KUKA KRL program: MyProgram_122().src

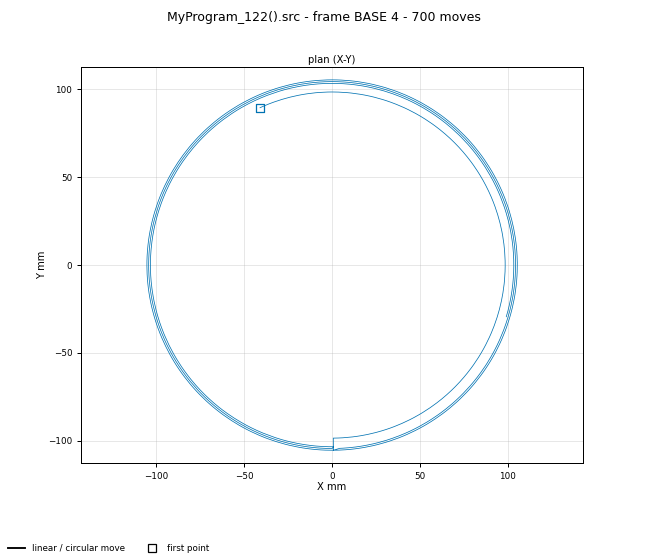
[picture p0: tool path of MyProgram_122().src in frame BASE 4, 700 of 700 moves have a stored position in this frame; points joined in program order, loops and branches not executed]
&ACCESS RVP
&REL 1
&PARAM TEMPLATE = C:\KRC\Roboter\Template\vorgabe
&PARAM EDITMASK = *
DEF MyProgram_122()
; ---- Setting reference (Base) ----
$BASE = BASE_DATA[4]

; --------------------------
; ---- Setting tool (TCP) ----
$TOOL = TOOL_DATA[3]
; --------------------------

$VEL.CP = VEL_APROX_PRINT
Startdeposition()
$VEL.CP = VEL_PRINT
LIN {X -40.9948,Y 89.481,Z 102,A 109.215,B 24.9184,C -2.0865,E1 24.9347,E2 -23.8628} C_DIS
LIN {X -38.5849,Y 90.5452,Z 102,A 107.7654,B 24.918,C -2.0917,E1 24.9383,E2 -22.4221} C_DIS
LIN {X -36.007,Y 91.6,Z 102,A 106.0596,B 24.918,C -2.091,E1 24.9428,E2 -20.711} C_DIS
LIN {X -33.1406,Y 92.6775,Z 102,A 104.2606,B 24.9179,C -2.0927,E1 24.9475,E2 -18.9123} C_DIS
LIN {X -30.6483,Y 93.5301,Z 102,A 102.9444,B 24.9171,C -2.1021,E1 24.9509,E2 -17.616} C_DIS
LIN {X -28.5659,Y 94.1882,Z 102,A 101.5499,B 24.9174,C -2.0993,E1 24.9547,E2 -16.2123} C_DIS
LIN {X -26.2518,Y 94.8593,Z 102,A 100.0341,B 24.9175,C -2.0968,E1 24.9588,E2 -14.6883} C_DIS
LIN {X -23.9044,Y 95.4778,Z 102,A 98.6262,B 24.9175,C -2.0984,E1 24.9626,E2 -13.2821} C_DIS
LIN {X -21.3156,Y 96.0877,Z 102,A 97.2954,B 24.9167,C -2.1074,E1 24.9661,E2 -11.9709} C_DIS
LIN {X -19.1831,Y 96.5372,Z 102,A 95.8048,B 24.9172,C -2.1007,E1 24.9703,E2 -10.4627} C_DIS
LIN {X -16.8179,Y 96.9772,Z 102,A 94.4012,B 24.9172,C -2.1016,E1 24.9741,E2 -9.06} C_DIS
LIN {X -14.1942,Y 97.3947,Z 102,A 92.9697,B 24.9168,C -2.1067,E1 24.978,E2 -7.6393} C_DIS
LIN {X -11.6809,Y 97.7276,Z 102,A 91.4888,B 24.9168,C -2.1075,E1 24.9821,E2 -6.159} C_DIS
LIN {X -9.5679,Y 97.9582,Z 102,A 90.1489,B 24.9169,C -2.1045,E1 24.9859,E2 -4.8112} C_DIS
LIN {X -7.202,Y 98.1607,Z 102,A 88.8601,B 24.9166,C -2.1084,E1 24.9895,E2 -3.5312} C_DIS
LIN {X -4.6001,Y 98.3161,Z 102,A 87.3398,B 24.9166,C -2.1088,E1 24.9937,E2 -2.0116} C_DIS
LIN {X -2.4401,Y 98.3944,Z 102,A 85.9895,B 24.9168,C -2.1059,E1 24.9975,E2 -0.6542} C_DIS
LIN {X -0.0607,Y 98.4244,Z 102,A 84.6864,B 24.9166,C -2.1091,E1 25.0011,E2 0.6413} C_DIS
LIN {X 3.6137,Y 98.3584,Z 102,A 82.4028,B 24.917,C -2.1042,E1 25.0075,E2 2.9361} C_DIS
LIN {X 6.3319,Y 98.2195,Z 102,A 81.0916,B 24.9162,C -2.1141,E1 25.0111,E2 4.2236} C_DIS
LIN {X 8.7012,Y 98.0382,Z 102,A 79.7032,B 24.9162,C -2.1138,E1 25.015,E2 5.6119} C_DIS
LIN {X 10.8611,Y 97.8236,Z 102,A 78.2118,B 24.9169,C -2.1054,E1 25.0191,E2 7.1222} C_DIS
LIN {X 13.4885,Y 97.4949,Z 102,A 76.8979,B 24.9162,C -2.1133,E1 25.0227,E2 8.4164} C_DIS
LIN {X 15.8676,Y 97.1361,Z 102,A 75.4989,B 24.9162,C -2.1129,E1 25.0266,E2 9.8148} C_DIS
LIN {X 18.2378,Y 96.7192,Z 102,A 73.8857,B 24.9169,C -2.1047,E1 25.0311,E2 11.4458} C_DIS
LIN {X 21.5808,Y 96.0296,Z 102,A 71.8924,B 24.917,C -2.1035,E1 25.0365,E2 13.4393} C_DIS
LIN {X 23.9252,Y 95.4726,Z 102,A 70.491,B 24.917,C -2.1027,E1 25.0403,E2 14.8406} C_DIS
LIN {X 26.4725,Y 94.7967,Z 102,A 69.0598,B 24.9169,C -2.1055,E1 25.0441,E2 16.2629} C_DIS
LIN {X 28.7857,Y 94.1201,Z 102,A 67.7784,B 24.9166,C -2.1089,E1 25.0476,E2 17.5339} C_DIS
LIN {X 30.9879,Y 93.4187,Z 102,A 66.2645,B 24.9172,C -2.1016,E1 25.0516,E2 19.0622} C_DIS
LIN {X 33.3777,Y 92.5912,Z 102,A 64.7955,B 24.9172,C -2.1004,E1 25.0555,E2 20.531} C_DIS
LIN {X 36.5486,Y 91.3873,Z 102,A 62.8757,B 24.9172,C -2.1004,E1 25.0605,E2 22.4465} C_DIS
LIN {X 38.7951,Y 90.4564,Z 102,A 61.3644,B 24.9177,C -2.0954,E1 25.0644,E2 23.9662} C_DIS
LIN {X 40.9951,Y 89.4809,Z 102,A 59.9392,B 24.9179,C -2.0929,E1 25.068,E2 25.3938} C_DIS
LIN {X 43.3728,Y 88.3516,Z 102,A 58.5388,B 24.9176,C -2.096,E1 25.0715,E2 26.7832} C_DIS
LIN {X 45.637,Y 87.2032,Z 102,A 57.1115,B 24.9176,C -2.096,E1 25.075,E2 28.2067} C_DIS
LIN {X 47.4644,Y 86.2239,Z 102,A 55.7597,B 24.9182,C -2.0889,E1 25.0784,E2 29.5713} C_DIS
LIN {X 50.0077,Y 84.7721,Z 102,A 54.0718,B 24.9183,C -2.0871,E1 25.0825,E2 31.2584} C_DIS
LIN {X 52.7518,Y 83.0937,Z 102,A 52.3478,B 24.9181,C -2.0898,E1 25.0865,E2 32.9706} C_DIS
LIN {X 54.8752,Y 81.7063,Z 102,A 50.9442,B 24.9181,C -2.0901,E1 25.0898,E2 34.3687} C_DIS
LIN {X 56.6984,Y 80.453,Z 102,A 49.5558,B 24.9185,C -2.0842,E1 25.093,E2 35.7664} C_DIS
LIN {X 58.6281,Y 79.058,Z 102,A 47.9451,B 24.9194,C -2.0733,E1 25.0967,E2 37.3971} C_DIS
LIN {X 61.4921,Y 76.8514,Z 102,A 45.8467,B 24.9197,C -2.0697,E1 25.1013,E2 39.4962} C_DIS
LIN {X 64.2951,Y 74.5223,Z 102,A 43.7362,B 24.92,C -2.066,E1 25.1058,E2 41.6072} C_DIS
LIN {X 66.9924,Y 72.1072,Z 102,A 41.6381,B 24.9203,C -2.0621,E1 25.1101,E2 43.7061} C_DIS
LIN {X 69.5959,Y 69.5978,Z 102,A 39.5415,B 24.9206,C -2.058,E1 25.1143,E2 45.8037} C_DIS
LIN {X 72.1053,Y 66.9944,Z 102,A 37.4476,B 24.9209,C -2.0537,E1 25.1183,E2 47.8985} C_DIS
LIN {X 74.5277,Y 64.2888,Z 102,A 35.3391,B 24.9213,C -2.0491,E1 25.1222,E2 50.0084} C_DIS
LIN {X 76.8501,Y 61.4937,Z 102,A 33.2405,B 24.9216,C -2.0448,E1 25.1259,E2 52.1075} C_DIS
LIN {X 79.0559,Y 58.631,Z 102,A 31.2593,B 24.9216,C -2.0443,E1 25.1292,E2 54.0804} C_DIS
LIN {X 80.4674,Y 56.6783,Z 102,A 29.6553,B 24.9225,C -2.033,E1 25.1318,E2 55.7032} C_DIS
LIN {X 82.6251,Y 53.4819,Z 102,A 27.8533,B 24.9216,C -2.0444,E1 25.1345,E2 57.4694} C_DIS
LIN {X 84.0971,Y 51.1345,Z 102,A 26.0418,B 24.9225,C -2.0325,E1 25.1372,E2 59.2998} C_DIS
LIN {X 85.7558,Y 48.3027,Z 102,A 24.1231,B 24.923,C -2.027,E1 25.1399,E2 61.2215} C_DIS
LIN {X 87.367,Y 45.326,Z 102,A 22.0924,B 24.9235,C -2.0192,E1 25.1426,E2 63.26} C_DIS
LIN {X 89.0655,Y 41.8874,Z 102,A 19.9181,B 24.9239,C -2.0152,E1 25.1452,E2 65.432} C_DIS
LIN {X 90.4636,Y 38.7786,Z 102,A 17.9782,B 24.9242,C -2.0112,E1 25.1474,E2 67.3707} C_DIS
LIN {X 91.6025,Y 36.0009,Z 102,A 16.2585,B 24.9245,C -2.0073,E1 25.1492,E2 69.0903} C_DIS
LIN {X 92.6741,Y 33.1502,Z 102,A 14.4811,B 24.9249,C -2.0018,E1 25.1509,E2 70.8706} C_DIS
LIN {X 93.5274,Y 30.6569,Z 102,A 13.1779,B 24.9245,C -2.0063,E1 25.152,E2 72.1558} C_DIS
LIN {X 94.1858,Y 28.574,Z 102,A 11.7748,B 24.9252,C -1.9973,E1 25.1532,E2 73.5722} C_DIS
LIN {X 94.8669,Y 26.2236,Z 102,A 10.2814,B 24.9257,C -1.9902,E1 25.1544,E2 75.0737} C_DIS
LIN {X 95.4791,Y 23.8988,Z 102,A 8.8903,B 24.926,C -1.9863,E1 25.1553,E2 76.4662} C_DIS
LIN {X 96.0936,Y 21.2884,Z 102,A 7.5866,B 24.9256,C -1.9916,E1 25.1561,E2 77.7497} C_DIS
LIN {X 96.5329,Y 19.2052,Z 102,A 6.0876,B 24.9267,C -1.9775,E1 25.157,E2 79.2733} C_DIS
LIN {X 96.9811,Y 16.795,Z 102,A 4.6967,B 24.9269,C -1.9744,E1 25.1577,E2 80.6632} C_DIS
LIN {X 97.3996,Y 14.1594,Z 102,A 3.3975,B 24.9265,C -1.9796,E1 25.1582,E2 81.9427} C_DIS
LIN {X 97.7073,Y 11.8542,Z 102,A 1.8366,B 24.9275,C -1.9671,E1 25.1588,E2 83.5237} C_DIS
LIN {X 98.1077,Y 7.8712,Z 102,A -0.4988,B 24.928,C -1.9595,E1 25.1594,E2 85.8633} C_DIS
LIN {X 98.316,Y 4.602,Z 102,A -2.3059,B 24.9282,C -1.9573,E1 25.1596,E2 87.6648} C_DIS
LIN {X 98.3951,Y 2.4176,Z 102,A -3.5706,B 24.9285,C -1.9535,E1 25.1598,E2 88.931} C_DIS
LIN {X 98.4213,Y -0.5653,Z 102,A -5.399,B 24.9291,C -1.9443,E1 25.1598,E2 90.7702} C_DIS
LIN {X 98.3552,Y -3.6891,Z 102,A -7.192,B 24.9295,C -1.9394,E1 25.1596,E2 92.564} C_DIS
LIN {X 98.2215,Y -6.3023,Z 102,A -8.4936,B 24.9292,C -1.9433,E1 25.1594,E2 93.8488} C_DIS
LIN {X 98.0389,Y -8.6932,Z 102,A -9.8785,B 24.9295,C -1.9392,E1 25.1591,E2 95.2351} C_DIS
LIN {X 97.8239,Y -10.8585,Z 102,A -11.3563,B 24.9304,C -1.9267,E1 25.1587,E2 96.7336} C_DIS
LIN {X 97.4984,Y -13.4641,Z 102,A -12.7946,B 24.9305,C -1.9254,E1 25.1582,E2 98.1666} C_DIS
LIN {X 97.1354,Y -15.8721,Z 102,A -14.0618,B 24.9305,C -1.9268,E1 25.1576,E2 99.423} C_DIS
LIN {X 96.7189,Y -18.2393,Z 102,A -15.5914,B 24.9311,C -1.9171,E1 25.1568,E2 100.9665} C_DIS
LIN {X 96.2873,Y -20.4005,Z 102,A -16.8444,B 24.9313,C -1.9142,E1 25.1561,E2 102.2191} C_DIS
LIN {X 95.7064,Y -22.9672,Z 102,A -18.2464,B 24.9313,C -1.9144,E1 25.1553,E2 103.6124} C_DIS
LIN {X 95.1162,Y -25.3005,Z 102,A -19.7578,B 24.9319,C -1.9056,E1 25.1542,E2 105.1358} C_DIS
LIN {X 94.4693,Y -27.6185,Z 102,A -21.1492,B 24.9322,C -1.9016,E1 25.1531,E2 106.5289} C_DIS
LIN {X 93.827,Y -29.731,Z 102,A -22.4266,B 24.9325,C -1.8978,E1 25.1521,E2 107.8078} C_DIS
LIN {X 92.9958,Y -32.2334,Z 102,A -23.9518,B 24.9328,C -1.8934,E1 25.1507,E2 109.3347} C_DIS
LIN {X 92.1626,Y -34.5434,Z 102,A -25.3693,B 24.9331,C -1.8895,E1 25.1493,E2 110.7536} C_DIS
LIN {X 91.3772,Y -36.5734,Z 102,A -26.6278,B 24.9333,C -1.8859,E1 25.1481,E2 112.0136} C_DIS
LIN {X 90.4568,Y -38.7942,Z 102,A -28.1186,B 24.9339,C -1.878,E1 25.1464,E2 113.5149} C_DIS
LIN {X 89.4819,Y -40.9929,Z 102,A -29.5106,B 24.9342,C -1.8741,E1 25.1448,E2 114.9085} C_DIS
LIN {X 88.3535,Y -43.3691,Z 102,A -30.9312,B 24.9342,C -1.8738,E1 25.1431,E2 116.3221} C_DIS
LIN {X 87.372,Y -45.3161,Z 102,A -32.2879,B 24.9347,C -1.8666,E1 25.1414,E2 117.6886} C_DIS
LIN {X 86.239,Y -47.4367,Z 102,A -33.6741,B 24.9349,C -1.863,E1 25.1395,E2 119.0761} C_DIS
LIN {X 84.9241,Y -49.7506,Z 102,A -35.2558,B 24.9353,C -1.8573,E1 25.1373,E2 120.6632} C_DIS
LIN {X 83.1402,Y -52.6793,Z 102,A -37.1049,B 24.9353,C -1.8573,E1 25.1346,E2 122.5028} C_DIS
LIN {X 81.7038,Y -54.8789,Z 102,A -38.5066,B 24.9353,C -1.858,E1 25.1324,E2 123.8958} C_DIS
LIN {X 80.4701,Y -56.6745,Z 102,A -39.8888,B 24.9358,C -1.85,E1 25.1302,E2 125.2902} C_DIS
LIN {X 79.0513,Y -58.6372,Z 102,A -41.503,B 24.9367,C -1.8382,E1 25.1275,E2 126.9245} C_DIS
LIN {X 76.8441,Y -61.5014,Z 102,A -43.4664,B 24.9367,C -1.8381,E1 25.1242,E2 128.8789} C_DIS
LIN {X 74.8272,Y -63.9373,Z 102,A -45.3366,B 24.9371,C -1.8321,E1 25.1208,E2 130.7546} C_DIS
LIN {X 72.5141,Y -66.5491,Z 102,A -47.3417,B 24.9374,C -1.828,E1 25.117,E2 132.7606} C_DIS
LIN {X 70.0204,Y -69.168,Z 102,A -49.3744,B 24.9375,C -1.8256,E1 25.1131,E2 134.7902} C_DIS
LIN {X 67.8252,Y -71.324,Z 102,A -51.305,B 24.9382,C -1.8158,E1 25.1092,E2 136.7358} C_DIS
LIN {X 65.2036,Y -73.7287,Z 102,A -53.3867,B 24.9386,C -1.8106,E1 25.1049,E2 138.8215} C_DIS
LIN {X 62.4378,Y -76.0852,Z 102,A -55.4885,B 24.9388,C -1.8063,E1 25.1003,E2 140.9253} C_DIS
LIN {X 59.5809,Y -78.3424,Z 102,A -57.5598,B 24.939,C -1.8036,E1 25.0958,E2 142.9953} C_DIS
LIN {X 57.4689,Y -79.9033,Z 102,A -58.9038,B 24.9388,C -1.8076,E1 25.0928,E2 144.3253} C_DIS
LIN {X 55.688,Y -81.1559,Z 102,A -60.2643,B 24.9392,C -1.8014,E1 25.0896,E2 145.6957} C_DIS
LIN {X 53.4819,Y -82.6251,Z 102,A -61.5838,B 24.9388,C -1.807,E1 25.0866,E2 146.9977} C_DIS
LIN {X 51.4301,Y -83.9176,Z 102,A -63.0217,B 24.939,C -1.8033,E1 25.0832,E2 148.4397} C_DIS
LIN {X 49.5184,Y -85.0606,Z 102,A -64.6107,B 24.94,C -1.7897,E1 25.0793,E2 150.0559} C_DIS
LIN {X 46.3754,Y -86.8143,Z 102,A -66.4863,B 24.9396,C -1.7944,E1 25.0747,E2 151.915} C_DIS
LIN {X 44.2425,Y -87.9205,Z 102,A -67.88,B 24.9398,C -1.7923,E1 25.0713,E2 153.3099} C_DIS
LIN {X 41.8786,Y -89.0696,Z 102,A -69.2882,B 24.9396,C -1.7945,E1 25.0677,E2 154.7093} C_DIS
LIN {X 39.6914,Y -90.0656,Z 102,A -70.8131,B 24.9401,C -1.7875,E1 25.0638,E2 156.2468} C_DIS
LIN {X 37.4486,Y -91.0209,Z 102,A -72.0962,B 24.9399,C -1.7906,E1 25.0606,E2 157.5196} C_DIS
LIN {X 35.4186,Y -91.8311,Z 102,A -73.4851,B 24.9403,C -1.7844,E1 25.0569,E2 158.9201} C_DIS
LIN {X 33.1106,Y -92.688,Z 102,A -75.0087,B 24.9407,C -1.7791,E1 25.0529,E2 160.453} C_DIS
LIN {X 30.6275,Y -93.5369,Z 102,A -76.318,B 24.9403,C -1.7854,E1 25.0495,E2 161.7448} C_DIS
LIN {X 28.004,Y -94.3549,Z 102,A -78.1162,B 24.9409,C -1.7761,E1 25.0446,E2 163.5618} C_DIS
LIN {X 24.8626,Y -95.2316,Z 102,A -79.8055,B 24.9405,C -1.7819,E1 25.0401,E2 165.2347} C_DIS
LIN {X 22.4912,Y -95.8193,Z 102,A -81.3437,B 24.9409,C -1.7762,E1 25.0359,E2 166.7843} C_DIS
LIN {X 20.3694,Y -96.2938,Z 102,A -82.8131,B 24.9415,C -1.7674,E1 25.0318,E2 168.2725} C_DIS
LIN {X 16.7828,Y -96.9831,Z 102,A -84.826,B 24.9413,C -1.7699,E1 25.0263,E2 170.2772} C_DIS
LIN {X 14.4201,Y -97.3626,Z 102,A -86.1187,B 24.9411,C -1.7726,E1 25.0228,E2 171.5623} C_DIS
LIN {X 11.5691,Y -97.7407,Z 102,A -87.6865,B 24.9409,C -1.7755,E1 25.0185,E2 173.122} C_DIS
LIN {X 8.2496,Y -98.0774,Z 102,A -89.6312,B 24.9409,C -1.7744,E1 25.0131,E2 175.0683} C_DIS
LIN {X 6.0869,Y -98.2361,Z 102,A -91.0704,B 24.9415,C -1.7673,E1 25.009,E2 176.5236} C_DIS
LIN {X 3.3973,Y -98.365,Z 102,A -92.4427,B 24.941,C -1.7739,E1 25.0052,E2 177.8798} C_DIS
LIN {X 0.6801,Y -98.4206,Z 102,A -93.8704,B 24.9407,C -1.7791,E1 25.0013,E2 179.295} C_DIS
Enddeposition()
LIN {X 0.7313,Y -105.3176,Z 103,A -93.556,B 24.9473,C -1.6774,E1 25.0015,E2 179.2217} C_DIS
Startdeposition()
$VEL.CP = VEL_PRINT
LIN {X -1.2925,Y -105.3149,Z 103,A -94.9939,B 24.9481,C -1.6637,E1 24.9974,E2 180.692} C_DIS
LIN {X -3.7589,Y -105.2551,Z 103,A -96.3407,B 24.9481,C -1.6634,E1 24.9936,E2 182.0398} C_DIS
LIN {X -6.3408,Y -105.1311,Z 103,A -97.7467,B 24.9481,C -1.6634,E1 24.9897,E2 183.4464} C_DIS
LIN {X -8.919,Y -104.9438,Z 103,A -99.1478,B 24.9481,C -1.6636,E1 24.9858,E2 184.8475} C_DIS
LIN {X -11.6089,Y -104.6811,Z 103,A -100.6185,B 24.9481,C -1.6636,E1 24.9817,E2 186.3187} C_DIS
LIN {X -14.1744,Y -104.3647,Z 103,A -102.0255,B 24.9481,C -1.6639,E1 24.9778,E2 187.7262} C_DIS
LIN {X -16.7314,Y -103.9854,Z 103,A -103.4327,B 24.9481,C -1.6642,E1 24.9739,E2 189.1339} C_DIS
LIN {X -19.2783,Y -103.5434,Z 103,A -104.8397,B 24.9481,C -1.6647,E1 24.9701,E2 190.5412} C_DIS
LIN {X -21.8136,Y -103.0391,Z 103,A -106.2476,B 24.9481,C -1.6652,E1 24.9662,E2 191.9495} C_DIS
LIN {X -24.2209,Y -102.4993,Z 103,A -107.5961,B 24.9481,C -1.6656,E1 24.9625,E2 193.2988} C_DIS
LIN {X -26.729,Y -101.874,Z 103,A -108.9991,B 24.948,C -1.6666,E1 24.9587,E2 194.7015} C_DIS
LIN {X -29.2211,Y -101.1874,Z 103,A -110.4124,B 24.948,C -1.6672,E1 24.9549,E2 196.1156} C_DIS
LIN {X -31.6604,Y -100.4507,Z 103,A -111.804,B 24.9479,C -1.668,E1 24.9512,E2 197.5077} C_DIS
LIN {X -34.2626,Y -99.594,Z 103,A -113.2888,B 24.9478,C -1.6694,E1 24.9473,E2 198.9919} C_DIS
LIN {X -36.5857,Y -98.7636,Z 103,A -114.6335,B 24.9478,C -1.6705,E1 24.9438,E2 200.3367} C_DIS
LIN {X -38.9985,Y -97.836,Z 103,A -116.0427,B 24.9476,C -1.6718,E1 24.9401,E2 201.746} C_DIS
LIN {X -41.3878,Y -96.8494,Z 103,A -117.4487,B 24.9476,C -1.6733,E1 24.9365,E2 203.1518} C_DIS
LIN {X -43.8595,Y -95.7561,Z 103,A -118.926,B 24.9474,C -1.6746,E1 24.9327,E2 204.6294} C_DIS
LIN {X -46.0901,Y -94.702,Z 103,A -120.2766,B 24.9474,C -1.6759,E1 24.9293,E2 205.9804} C_DIS
LIN {X -48.4003,Y -93.5423,Z 103,A -121.6818,B 24.9473,C -1.6777,E1 24.9258,E2 207.385} C_DIS
LIN {X -50.6814,Y -92.3263,Z 103,A -123.0919,B 24.9471,C -1.6794,E1 24.9223,E2 208.7951} C_DIS
LIN {X -52.9319,Y -91.0548,Z 103,A -124.5028,B 24.9471,C -1.6812,E1 24.9189,E2 210.2059} C_DIS
LIN {X -55.1506,Y -89.7283,Z 103,A -125.9134,B 24.9469,C -1.6832,E1 24.9156,E2 211.6163} C_DIS
LIN {X -57.3091,Y -88.3651,Z 103,A -127.3087,B 24.9468,C -1.6851,E1 24.9123,E2 213.0115} C_DIS
LIN {X -59.5845,Y -86.8481,Z 103,A -128.8,B 24.9466,C -1.6873,E1 24.9088,E2 214.5024} C_DIS
LIN {X -61.602,Y -85.4281,Z 103,A -130.1469,B 24.9466,C -1.6894,E1 24.9058,E2 215.849} C_DIS
LIN {X -63.6799,Y -83.8906,Z 103,A -131.5635,B 24.9464,C -1.6915,E1 24.9026,E2 217.2657} C_DIS
LIN {X -65.7195,Y -82.3025,Z 103,A -132.9703,B 24.9462,C -1.694,E1 24.8995,E2 218.6716} C_DIS
LIN {X -67.7195,Y -80.6649,Z 103,A -134.3826,B 24.9461,C -1.6965,E1 24.8965,E2 220.0835} C_DIS
LIN {X -69.6787,Y -78.9787,Z 103,A -135.7996,B 24.9459,C -1.6988,E1 24.8935,E2 221.5005} C_DIS
LIN {X -71.6828,Y -77.1652,Z 103,A -137.2715,B 24.9457,C -1.7017,E1 24.8905,E2 222.9715} C_DIS
LIN {X -73.555,Y -75.3828,Z 103,A -138.684,B 24.9456,C -1.7044,E1 24.8876,E2 224.3835} C_DIS
LIN {X -75.3,Y -73.6388,Z 103,A -140.0112,B 24.9453,C -1.7078,E1 24.885,E2 225.7082} C_DIS
LIN {X -77.0845,Y -71.7687,Z 103,A -141.4455,B 24.9453,C -1.7099,E1 24.8823,E2 227.1438} C_DIS
LIN {X -78.8226,Y -69.8553,Z 103,A -142.8635,B 24.945,C -1.7126,E1 24.8796,E2 228.5617} C_DIS
LIN {X -80.5896,Y -67.8102,Z 103,A -144.3363,B 24.9448,C -1.7159,E1 24.877,E2 230.0333} C_DIS
LIN {X -82.2294,Y -65.812,Z 103,A -145.7499,B 24.9446,C -1.7189,E1 24.8745,E2 231.4463} C_DIS
LIN {X -83.6473,Y -63.998,Z 103,A -147.0343,B 24.9446,C -1.7208,E1 24.8723,E2 232.7323} C_DIS
LIN {X -85.3596,Y -61.6979,Z 103,A -148.5772,B 24.9442,C -1.7253,E1 24.8697,E2 234.2721} C_DIS
LIN {X -86.8481,Y -59.5845,Z 103,A -149.9913,B 24.944,C -1.7285,E1 24.8675,E2 235.6853} C_DIS
LIN {X -88.2842,Y -57.4352,Z 103,A -151.4054,B 24.9438,C -1.7319,E1 24.8653,E2 237.0986} C_DIS
LIN {X -89.6671,Y -55.2513,Z 103,A -152.8199,B 24.9436,C -1.7352,E1 24.8632,E2 238.5122} C_DIS
LIN {X -90.9961,Y -53.0341,Z 103,A -154.2342,B 24.9433,C -1.7387,E1 24.8612,E2 239.9256} C_DIS
LIN {X -92.2702,Y -50.785,Z 103,A -155.6485,B 24.9431,C -1.7422,E1 24.8593,E2 241.3389} C_DIS
LIN {X -93.4887,Y -48.5052,Z 103,A -157.0636,B 24.9429,C -1.7458,E1 24.8574,E2 242.7532} C_DIS
LIN {X -94.5986,Y -46.3019,Z 103,A -158.3982,B 24.9426,C -1.7498,E1 24.8558,E2 244.0853} C_DIS
LIN {X -95.7561,Y -43.8595,Z 103,A -159.8931,B 24.9424,C -1.753,E1 24.854,E2 245.5806} C_DIS
LIN {X -96.7566,Y -41.6044,Z 103,A -161.2487,B 24.9422,C -1.7564,E1 24.8525,E2 246.9356} C_DIS
LIN {X -97.7929,Y -39.1082,Z 103,A -162.7234,B 24.9419,C -1.7605,E1 24.8509,E2 248.4088} C_DIS
LIN {X -99.1661,Y -35.4822,Z 103,A -164.8465,B 24.9415,C -1.7662,E1 24.8489,E2 250.5302} C_DIS
LIN {X -99.9693,Y -33.1495,Z 103,A -166.1975,B 24.9413,C -1.7699,E1 24.8477,E2 251.88} C_DIS
LIN {X -100.7876,Y -30.5736,Z 103,A -167.6771,B 24.941,C -1.774,E1 24.8464,E2 253.3585} C_DIS
LIN {X -101.5076,Y -28.0909,Z 103,A -169.0929,B 24.9408,C -1.778,E1 24.8454,E2 254.773} C_DIS
LIN {X -102.4448,Y -24.4502,Z 103,A -171.157,B 24.9404,C -1.7836,E1 24.844,E2 256.8358} C_DIS
LIN {X -103.014,Y -21.9287,Z 103,A -172.5495,B 24.94,C -1.7885,E1 24.8431,E2 258.2249} C_DIS
LIN {X -103.706,Y -18.3741,Z 103,A -174.5824,B 24.9398,C -1.7924,E1 24.8421,E2 260.2604} C_DIS
LIN {X -104.1649,Y -15.5705,Z 103,A -176.1126,B 24.9394,C -1.7978,E1 24.8414,E2 261.7869} C_DIS
LIN {X -104.5156,Y -13.0095,Z 103,A -177.5287,B 24.9391,C -1.8019,E1 24.8409,E2 263.2017} C_DIS
LIN {X -104.8034,Y -10.4406,Z 103,A -178.9447,B 24.9389,C -1.806,E1 24.8405,E2 264.6162} C_DIS
LIN {X -105.0374,Y -7.748,Z 103,A 179.5798,B 24.9386,C -1.8105,E1 24.8402,E2 266.0899} C_DIS
LIN {X -105.196,Y -5.1679,Z 103,A 178.1638,B 24.9383,C -1.8147,E1 24.8399,E2 267.5045} C_DIS
LIN {X -105.2911,Y -2.5848,Z 103,A 176.7475,B 24.938,C -1.8189,E1 24.8399,E2 268.9193} C_DIS
LIN {X -105.3199,Y -0.4985,Z 103,A 175.5316,B 24.938,C -1.8197,E1 24.8398,E2 270.1407} C_DIS
LIN {X -105.2946,Y 2.394,Z 103,A 174.0149,B 24.9374,C -1.8268,E1 24.8398,E2 271.6496} C_DIS
LIN {X -105.196,Y 5.1679,Z 103,A 172.4989,B 24.9371,C -1.8314,E1 24.84,E2 273.1637} C_DIS
LIN {X -105.0374,Y 7.748,Z 103,A 171.083,B 24.9368,C -1.8356,E1 24.8403,E2 274.5781} C_DIS
LIN {X -104.7054,Y 11.3769,Z 103,A 169.0769,B 24.9365,C -1.8412,E1 24.8408,E2 276.5829} C_DIS
LIN {X -104.3647,Y 14.1744,Z 103,A 167.5426,B 24.9361,C -1.8461,E1 24.8414,E2 278.1147} C_DIS
LIN {X -104.0034,Y 16.6149,Z 103,A 166.1908,B 24.9358,C -1.8501,E1 24.8419,E2 279.465} C_DIS
LIN {X -103.5434,Y 19.2783,Z 103,A 164.7104,B 24.9355,C -1.8544,E1 24.8427,E2 280.9438} C_DIS
LIN {X -103.0391,Y 21.8136,Z 103,A 163.294,B 24.9352,C -1.8585,E1 24.8435,E2 282.3587} C_DIS
LIN {X -102.4993,Y 24.2209,Z 103,A 161.9772,B 24.9349,C -1.8637,E1 24.8443,E2 283.6709} C_DIS
LIN {X -101.5383,Y 27.9772,Z 103,A 159.8433,B 24.9345,C -1.8696,E1 24.8458,E2 285.8034} C_DIS
LIN {X -100.8212,Y 30.4606,Z 103,A 158.3975,B 24.9343,C -1.8726,E1 24.8469,E2 287.2503} C_DIS
LIN {X -100.007,Y 33.0378,Z 103,A 156.9221,B 24.934,C -1.877,E1 24.8482,E2 288.7235} C_DIS
LIN {X -99.2051,Y 35.371,Z 103,A 155.5659,B 24.9337,C -1.8807,E1 24.8495,E2 290.0787} C_DIS
LIN {X -98.2654,Y 37.9052,Z 103,A 154.0907,B 24.9334,C -1.885,E1 24.8509,E2 291.5518} C_DIS
LIN {X -97.3056,Y 40.3053,Z 103,A 152.675,B 24.9331,C -1.889,E1 24.8524,E2 292.9659} C_DIS
LIN {X -96.2871,Y 42.6812,Z 103,A 151.2592,B 24.9328,C -1.8929,E1 24.854,E2 294.3802} C_DIS
LIN {X -95.2604,Y 44.9245,Z 103,A 149.9034,B 24.9326,C -1.8965,E1 24.8556,E2 295.7348} C_DIS
LIN {X -94.0769,Y 47.3543,Z 103,A 148.4286,B 24.9323,C -1.9007,E1 24.8574,E2 297.2076} C_DIS
LIN {X -92.9413,Y 49.5446,Z 103,A 147.0725,B 24.932,C -1.9042,E1 24.8591,E2 298.5626} C_DIS
LIN {X -91.6975,Y 51.8105,Z 103,A 145.6575,B 24.9318,C -1.908,E1 24.8611,E2 299.976} C_DIS
LIN {X -90.3384,Y 54.1467,Z 103,A 144.183,B 24.9315,C -1.912,E1 24.8632,E2 301.4485} C_DIS
LIN {X -88.9824,Y 56.3475,Z 103,A 142.7677,B 24.9312,C -1.9157,E1 24.8652,E2 302.8622} C_DIS
LIN {X -87.6376,Y 58.4158,Z 103,A 141.4175,B 24.9309,C -1.9192,E1 24.8673,E2 304.2109} C_DIS
LIN {X -86.1103,Y 60.6457,Z 103,A 139.9381,B 24.9307,C -1.9229,E1 24.8697,E2 305.6887} C_DIS
LIN {X -84.6657,Y 62.6457,Z 103,A 138.588,B 24.9304,C -1.9263,E1 24.8719,E2 307.0373} C_DIS
LIN {X -83.0588,Y 64.7616,Z 103,A 137.1355,B 24.9302,C -1.9299,E1 24.8744,E2 308.4882} C_DIS
LIN {X -81.4898,Y 66.7245,Z 103,A 135.7592,B 24.9299,C -1.9332,E1 24.8768,E2 309.8631} C_DIS
LIN {X -79.8278,Y 68.7043,Z 103,A 134.3402,B 24.9297,C -1.9363,E1 24.8793,E2 311.281} C_DIS
LIN {X -78.0391,Y 70.7305,Z 103,A 132.8663,B 24.9294,C -1.9399,E1 24.8821,E2 312.7528} C_DIS
LIN {X -76.2797,Y 72.6243,Z 103,A 131.4527,B 24.9292,C -1.9432,E1 24.8848,E2 314.165} C_DIS
LIN {X -74.4745,Y 74.4745,Z 103,A 130.039,B 24.929,C -1.9463,E1 24.8875,E2 315.5772} C_DIS
LIN {X -72.7092,Y 76.198,Z 103,A 128.6899,B 24.9288,C -1.9493,E1 24.8903,E2 316.9248} C_DIS
LIN {X -70.8173,Y 77.9594,Z 103,A 127.2766,B 24.9285,C -1.9523,E1 24.8932,E2 318.3367} C_DIS
LIN {X -68.8831,Y 79.6736,Z 103,A 125.8585,B 24.9283,C -1.955,E1 24.8961,E2 319.7538} C_DIS
LIN {X -66.9545,Y 81.3006,Z 103,A 124.4838,B 24.9281,C -1.958,E1 24.8991,E2 321.1267} C_DIS
LIN {X -64.7979,Y 83.0309,Z 103,A 122.9728,B 24.9279,C -1.961,E1 24.9024,E2 322.6362} C_DIS
LIN {X -62.7407,Y 84.5961,Z 103,A 121.5602,B 24.9277,C -1.9637,E1 24.9055,E2 324.0474} C_DIS
LIN {X -60.6457,Y 86.1103,Z 103,A 120.1477,B 24.9275,C -1.9663,E1 24.9087,E2 325.4585} C_DIS
LIN {X -57.6507,Y 88.1421,Z 103,A 118.1487,B 24.9273,C -1.9691,E1 24.9134,E2 327.4576} C_DIS
LIN {X -55.3512,Y 89.6047,Z 103,A 116.6768,B 24.9271,C -1.9723,E1 24.9169,E2 328.9266} C_DIS
LIN {X -53.3457,Y 90.8119,Z 103,A 115.3635,B 24.9271,C -1.9731,E1 24.92,E2 330.2418} C_DIS
LIN {X -50.785,Y 92.2702,Z 103,A 113.7942,B 24.9267,C -1.9772,E1 24.9238,E2 331.8062} C_DIS
LIN {X -48.5052,Y 93.4887,Z 103,A 112.3824,B 24.9265,C -1.9793,E1 24.9273,E2 333.2167} C_DIS
LIN {X -46.3019,Y 94.5986,Z 103,A 111.0489,B 24.9264,C -1.9818,E1 24.9306,E2 334.5479} C_DIS
LIN {X -43.8595,Y 95.7561,Z 103,A 109.5605,B 24.9262,C -1.9834,E1 24.9344,E2 336.0362} C_DIS
LIN {X -41.4963,Y 96.8037,Z 103,A 108.1497,B 24.9262,C -1.9853,E1 24.938,E2 337.4459} C_DIS
LIN {X -39.1082,Y 97.7929,Z 103,A 106.7391,B 24.926,C -1.9871,E1 24.9417,E2 338.8553} C_DIS
LIN {X -36.6964,Y 98.7232,Z 103,A 105.3289,B 24.9258,C -1.9888,E1 24.9453,E2 340.2643} C_DIS
LIN {X -34.2626,Y 99.594,Z 103,A 103.9188,B 24.9258,C -1.9904,E1 24.949,E2 341.6734} C_DIS
LIN {X -31.9202,Y 100.3686,Z 103,A 102.5682,B 24.9256,C -1.9917,E1 24.9526,E2 343.0234} C_DIS
LIN {X -29.4474,Y 101.1217,Z 103,A 101.172,B 24.9255,C -1.9936,E1 24.9564,E2 344.4173} C_DIS
LIN {X -26.8432,Y 101.8447,Z 103,A 99.6899,B 24.9254,C -1.9947,E1 24.9604,E2 345.8992} C_DIS
LIN {X -24.4502,Y 102.4448,Z 103,A 98.3754,B 24.9252,C -1.997,E1 24.9639,E2 347.21} C_DIS
LIN {X -21.9287,Y 103.014,Z 103,A 96.9361,B 24.9252,C -1.997,E1 24.9678,E2 348.6511} C_DIS
LIN {X -19.394,Y 103.5212,Z 103,A 95.5273,B 24.9252,C -1.9981,E1 24.9717,E2 350.059} C_DIS
LIN {X -16.7314,Y 103.9854,Z 103,A 94.0547,B 24.9251,C -1.999,E1 24.9757,E2 351.5307} C_DIS
LIN {X -14.1744,Y 104.3647,Z 103,A 92.6465,B 24.9251,C -1.9999,E1 24.9796,E2 352.938} C_DIS
LIN {X -11.6089,Y 104.6811,Z 103,A 91.2386,B 24.925,C -2.0006,E1 24.9835,E2 354.3451} C_DIS
LIN {X -8.1224,Y 105.0075,Z 103,A 89.3002,B 24.925,C -2.0003,E1 24.9889,E2 356.2852} C_DIS
LIN {X -5.1679,Y 105.196,Z 103,A 87.7195,B 24.9249,C -2.002,E1 24.9933,E2 357.8623} C_DIS
LIN {X -2.8306,Y 105.2835,Z 103,A 86.435,B 24.9249,C -2.002,E1 24.9969,E2 359.1471} C_DIS
LIN {X -0.1178,Y 105.3221,Z 103,A 84.9645,B 24.9249,C -2.0024,E1 25.001,E2 360.6165} C_DIS
LIN {X 2.5848,Y 105.2911,Z 103,A 83.4989,B 24.9248,C -2.0028,E1 25.0051,E2 362.0809} C_DIS
LIN {X 5.1679,Y 105.196,Z 103,A 82.0921,B 24.9248,C -2.0028,E1 25.009,E2 363.4872} C_DIS
LIN {X 7.748,Y 105.0374,Z 103,A 80.6859,B 24.9248,C -2.0028,E1 25.013,E2 364.8929} C_DIS
LIN {X 10.2061,Y 104.8265,Z 103,A 79.339,B 24.9248,C -2.0025,E1 25.0167,E2 366.2397} C_DIS
LIN {X 12.601,Y 104.5649,Z 103,A 78.0251,B 24.9248,C -2.0022,E1 25.0203,E2 367.5534} C_DIS
LIN {X 15.3374,Y 104.1994,Z 103,A 76.528,B 24.9248,C -2.002,E1 25.0245,E2 369.0497} C_DIS
LIN {X 18.0062,Y 103.7722,Z 103,A 75.0638,B 24.9248,C -2.0017,E1 25.0285,E2 370.5131} C_DIS
LIN {X 20.4318,Y 103.3213,Z 103,A 73.7178,B 24.9249,C -2.001,E1 25.0322,E2 371.8592} C_DIS
LIN {X 23.0764,Y 102.7637,Z 103,A 72.2541,B 24.9249,C -2.0005,E1 25.0362,E2 373.3221} C_DIS
LIN {X 25.5914,Y 102.1664,Z 103,A 70.8496,B 24.925,C -1.9998,E1 25.04,E2 374.7263} C_DIS
LIN {X 27.9772,Y 101.5383,Z 103,A 69.5043,B 24.925,C -1.9988,E1 25.0436,E2 376.0718} C_DIS
LIN {X 30.4606,Y 100.8212,Z 103,A 68.1265,B 24.925,C -1.9989,E1 25.0473,E2 377.447} C_DIS
LIN {X 33.0378,Y 100.007,Z 103,A 66.6375,B 24.9252,C -1.997,E1 25.0513,E2 378.9378} C_DIS
LIN {X 35.371,Y 99.2051,Z 103,A 65.2979,B 24.9253,C -1.9959,E1 25.0548,E2 380.2772} C_DIS
LIN {X 37.795,Y 98.3072,Z 103,A 63.8897,B 24.9254,C -1.9945,E1 25.0585,E2 381.6857} C_DIS
LIN {X 41.3878,Y 96.8494,Z 103,A 61.7851,B 24.9256,C -1.9925,E1 25.0639,E2 383.7903} C_DIS
LIN {X 43.7521,Y 95.8045,Z 103,A 60.3873,B 24.9256,C -1.9912,E1 25.0675,E2 385.1876} C_DIS
LIN {X 46.0901,Y 94.702,Z 103,A 58.9798,B 24.9258,C -1.9894,E1 25.071,E2 386.5956} C_DIS
LIN {X 48.5052,Y 93.4887,Z 103,A 57.5187,B 24.9259,C -1.9879,E1 25.0747,E2 388.0564} C_DIS
LIN {X 50.785,Y 92.2702,Z 103,A 56.1166,B 24.926,C -1.9861,E1 25.0781,E2 389.4586} C_DIS
LIN {X 53.0341,Y 90.9961,Z 103,A 54.7145,B 24.9262,C -1.9843,E1 25.0815,E2 390.8609} C_DIS
LIN {X 54.8577,Y 89.9063,Z 103,A 53.5023,B 24.9265,C -1.9803,E1 25.0844,E2 392.0787} C_DIS
LIN {X 57.336,Y 88.3478,Z 103,A 51.9752,B 24.9265,C -1.9804,E1 25.088,E2 393.6005} C_DIS
LIN {X 59.5845,Y 86.8481,Z 103,A 50.5101,B 24.9266,C -1.9782,E1 25.0914,E2 395.066} C_DIS
LIN {X 61.602,Y 85.4281,Z 103,A 49.1729,B 24.9268,C -1.9761,E1 25.0944,E2 396.4034} C_DIS
LIN {X 63.6799,Y 83.8906,Z 103,A 47.8027,B 24.9268,C -1.9751,E1 25.0975,E2 397.7711} C_DIS
LIN {X 65.812,Y 82.2294,Z 103,A 46.3078,B 24.9271,C -1.9714,E1 25.1008,E2 399.2693} C_DIS
LIN {X 67.7195,Y 80.6649,Z 103,A 44.9711,B 24.9273,C -1.9691,E1 25.1036,E2 400.6063} C_DIS
LIN {X 69.6788,Y 78.9787,Z 103,A 43.5657,B 24.9275,C -1.9663,E1 25.1066,E2 402.0127} C_DIS
LIN {X 71.6828,Y 77.1652,Z 103,A 42.107,B 24.9277,C -1.9638,E1 25.1096,E2 403.4714} C_DIS
LIN {X 73.555,Y 75.3828,Z 103,A 40.707,B 24.9279,C -1.9611,E1 25.1124,E2 404.872} C_DIS
LIN {X 75.3,Y 73.6388,Z 103,A 39.3824,B 24.9281,C -1.959,E1 25.115,E2 406.196} C_DIS
LIN {X 77.0845,Y 71.7686,Z 103,A 37.9666,B 24.9283,C -1.9555,E1 25.1177,E2 407.6139} C_DIS
LIN {X 78.8226,Y 69.8553,Z 103,A 36.5957,B 24.9284,C -1.9537,E1 25.1203,E2 408.9828} C_DIS
LIN {X 80.5896,Y 67.8102,Z 103,A 35.1093,B 24.9287,C -1.9496,E1 25.123,E2 410.4721} C_DIS
LIN {X 82.2294,Y 65.812,Z 103,A 33.7104,B 24.929,C -1.9466,E1 25.1255,E2 411.8717} C_DIS
LIN {X 83.7479,Y 63.8675,Z 103,A 32.375,B 24.9292,C -1.9436,E1 25.1277,E2 413.2078} C_DIS
LIN {X 85.29,Y 61.7929,Z 103,A 30.9716,B 24.9294,C -1.9402,E1 25.1301,E2 414.6125} C_DIS
LIN {X 86.7808,Y 59.6812,Z 103,A 29.5779,B 24.9296,C -1.9372,E1 25.1323,E2 416.0064} C_DIS
LIN {X 88.2842,Y 57.4352,Z 103,A 28.1156,B 24.9299,C -1.9337,E1 25.1345,E2 417.4697} C_DIS
LIN {X 89.6047,Y 55.3512,Z 103,A 26.7811,B 24.9301,C -1.9305,E1 25.1365,E2 418.805} C_DIS
LIN {X 90.9361,Y 53.1355,Z 103,A 25.3781,B 24.9304,C -1.9269,E1 25.1385,E2 420.2094} C_DIS
LIN {X 92.2127,Y 50.8878,Z 103,A 23.9801,B 24.9306,C -1.9234,E1 25.1404,E2 421.6082} C_DIS
LIN {X 94.0233,Y 47.4593,Z 103,A 21.8883,B 24.931,C -1.9183,E1 25.1431,E2 423.7011} C_DIS
LIN {X 95.1597,Y 45.1375,Z 103,A 20.4856,B 24.9313,C -1.9145,E1 25.1448,E2 425.1053} C_DIS
LIN {X 96.2871,Y 42.6812,Z 103,A 19.0292,B 24.9315,C -1.9109,E1 25.1465,E2 426.5623} C_DIS
LIN {X 97.3056,Y 40.3053,Z 103,A 17.6319,B 24.9318,C -1.9072,E1 25.148,E2 427.9607} C_DIS
LIN {X 98.2654,Y 37.9052,Z 103,A 16.2346,B 24.9321,C -1.9034,E1 25.1495,E2 429.3591} C_DIS
LIN {X 99.1661,Y 35.4822,Z 103,A 14.8372,B 24.9324,C -1.8996,E1 25.1508,E2 430.7577} C_DIS
LIN {X 99.9693,Y 33.1495,Z 103,A 13.5037,B 24.9326,C -1.896,E1 25.152,E2 432.0922} C_DIS
LIN {X 100.7528,Y 30.6861,Z 103,A 12.1018,B 24.9329,C -1.8919,E1 25.1532,E2 433.4957} C_DIS
LIN {X 101.5076,Y 28.0909,Z 103,A 10.6461,B 24.9332,C -1.888,E1 25.1543,E2 434.9523} C_DIS
LIN {X 102.1371,Y 25.7055,Z 103,A 9.3078,B 24.9335,C -1.8841,E1 25.1552,E2 436.2921} C_DIS
LIN {X 102.7637,Y 23.0764,Z 103,A 7.8523,B 24.9337,C -1.8801,E1 25.1561,E2 437.7485} C_DIS
LIN {X 103.2754,Y 20.6629,Z 103,A 6.514,B 24.934,C -1.8761,E1 25.1569,E2 439.0885} C_DIS
LIN {X 103.7514,Y 18.1222,Z 103,A 5.1224,B 24.9343,C -1.8723,E1 25.1576,E2 440.4809} C_DIS
LIN {X 104.1238,Y 15.836,Z 103,A 3.8968,B 24.9345,C -1.8698,E1 25.1581,E2 441.7052} C_DIS
LIN {X 104.5156,Y 13.0095,Z 103,A 2.324,B 24.9349,C -1.864,E1 25.1587,E2 443.2824} C_DIS
LIN {X 104.8034,Y 10.4406,Z 103,A 0.9326,B 24.9351,C -1.8601,E1 25.1591,E2 444.6747} C_DIS
LIN {X 105.0374,Y 7.748,Z 103,A -0.5276,B 24.9354,C -1.8558,E1 25.1594,E2 446.1364} C_DIS
LIN {X 105.196,Y 5.1679,Z 103,A -1.9242,B 24.9357,C -1.8517,E1 25.1596,E2 447.5343} C_DIS
LIN {X 105.3127,Y 1.4103,Z 103,A -3.9505,B 24.9361,C -1.8459,E1 25.1598,E2 449.5623} C_DIS
LIN {X 105.3127,Y -1.4103,Z 103,A -5.4207,B 24.9363,C -1.8437,E1 25.1598,E2 451.029} C_DIS
LIN {X 105.2551,Y -3.7589,Z 103,A -6.753,B 24.9367,C -1.8373,E1 25.1596,E2 452.3686} C_DIS
LIN {X 105.1311,Y -6.3408,Z 103,A -8.1494,B 24.937,C -1.8331,E1 25.1594,E2 453.7663} C_DIS
LIN {X 104.9438,Y -8.919,Z 103,A -9.5406,B 24.9373,C -1.8292,E1 25.1591,E2 455.1586} C_DIS
LIN {X 104.6811,Y -11.6089,Z 103,A -11.0007,B 24.9376,C -1.8249,E1 25.1587,E2 456.6203} C_DIS
LIN {X 104.3647,Y -14.1744,Z 103,A -12.3975,B 24.9379,C -1.8207,E1 25.1582,E2 458.0186} C_DIS
LIN {X 103.9997,Y -16.6386,Z 103,A -13.7463,B 24.9381,C -1.8166,E1 25.1576,E2 459.3691} C_DIS
LIN {X 103.5434,Y -19.2783,Z 103,A -15.1902,B 24.9384,C -1.8125,E1 25.1569,E2 460.8143} C_DIS
LIN {X 103.0391,Y -21.8136,Z 103,A -16.587,B 24.9387,C -1.8084,E1 25.1561,E2 462.2126} C_DIS
LIN {X 102.4993,Y -24.2209,Z 103,A -17.9248,B 24.939,C -1.8043,E1 25.1553,E2 463.5524} C_DIS
LIN {X 101.5383,Y -27.9772,Z 103,A -20.0147,B 24.9394,C -1.7984,E1 25.1538,E2 465.6442} C_DIS
LIN {X 100.7876,Y -30.5736,Z 103,A -21.475,B 24.9397,C -1.7941,E1 25.1527,E2 467.1061} C_DIS
LIN {X 100.007,Y -33.0378,Z 103,A -22.8718,B 24.9399,C -1.7901,E1 25.1515,E2 468.5045} C_DIS
LIN {X 99.2051,Y -35.371,Z 103,A -24.205,B 24.9402,C -1.7863,E1 25.1502,E2 469.8391} C_DIS
LIN {X 98.3072,Y -37.795,Z 103,A -25.6019,B 24.9405,C -1.7824,E1 25.1489,E2 471.2376} C_DIS
LIN {X 97.35,Y -40.1962,Z 103,A -26.9985,B 24.9407,C -1.7784,E1 25.1474,E2 472.6358} C_DIS
LIN {X 96.4423,Y -42.3253,Z 103,A -28.2939,B 24.9411,C -1.7731,E1 25.1459,E2 473.9368} C_DIS
LIN {X 95.2604,Y -44.9245,Z 103,A -29.7927,B 24.9412,C -1.7706,E1 25.1442,E2 475.4332} C_DIS
LIN {X 94.0769,Y -47.3543,Z 103,A -31.2535,B 24.9415,C -1.7666,E1 25.1424,E2 476.8956} C_DIS
LIN {X 93.0625,Y -49.3146,Z 103,A -32.4781,B 24.9418,C -1.7621,E1 25.1408,E2 478.1244} C_DIS
LIN {X 91.6975,Y -51.8105,Z 103,A -33.9845,B 24.942,C -1.7593,E1 25.1387,E2 479.6296} C_DIS
LIN {X 90.3983,Y -54.0453,Z 103,A -35.3819,B 24.9422,C -1.7556,E1 25.1368,E2 481.0285} C_DIS
LIN {X 89.0448,Y -56.2475,Z 103,A -36.7795,B 24.9425,C -1.7519,E1 25.1347,E2 482.4278} C_DIS
LIN {X 87.6376,Y -58.4159,Z 103,A -38.1821,B 24.9427,C -1.7481,E1 25.1325,E2 483.8323} C_DIS
LIN {X 86.1776,Y -60.549,Z 103,A -39.5523,B 24.9429,C -1.7457,E1 25.1304,E2 485.2015} C_DIS
LIN {X 84.6657,Y -62.6457,Z 103,A -40.9731,B 24.9432,C -1.7412,E1 25.128,E2 486.6259} C_DIS
LIN {X 83.0309,Y -64.7979,Z 103,A -42.4347,B 24.9434,C -1.7376,E1 25.1255,E2 488.0892} C_DIS
LIN {X 81.4898,Y -66.7245,Z 103,A -43.7693,B 24.9436,C -1.7344,E1 25.1232,E2 489.4252} C_DIS
LIN {X 79.8278,Y -68.7043,Z 103,A -45.1675,B 24.9438,C -1.731,E1 25.1207,E2 490.8249} C_DIS
LIN {X 78.0391,Y -70.7305,Z 103,A -46.6298,B 24.9441,C -1.7276,E1 25.1179,E2 492.2888} C_DIS
LIN {X 76.2797,Y -72.6244,Z 103,A -48.0283,B 24.9443,C -1.7244,E1 25.1153,E2 493.6888} C_DIS
LIN {X 74.4745,Y -74.4745,Z 103,A -49.4271,B 24.9445,C -1.7212,E1 25.1125,E2 495.0891} C_DIS
LIN {X 72.7092,Y -76.198,Z 103,A -50.7622,B 24.9447,C -1.7183,E1 25.1098,E2 496.4256} C_DIS
LIN {X 70.8173,Y -77.9594,Z 103,A -52.1614,B 24.9449,C -1.7153,E1 25.1069,E2 497.8263} C_DIS
LIN {X 68.794,Y -79.7514,Z 103,A -53.6244,B 24.9451,C -1.7122,E1 25.1039,E2 499.2908} C_DIS
LIN {X 67.0031,Y -81.2602,Z 103,A -54.9113,B 24.9453,C -1.7088,E1 25.1011,E2 500.5807} C_DIS
LIN {X 64.907,Y -82.9447,Z 103,A -56.3494,B 24.9454,C -1.7066,E1 25.098,E2 502.0186} C_DIS
LIN {X 62.7407,Y -84.5961,Z 103,A -57.8234,B 24.9456,C -1.7038,E1 25.0947,E2 503.4939} C_DIS
LIN {X 60.6457,Y -86.1103,Z 103,A -59.2232,B 24.9458,C -1.7011,E1 25.0915,E2 504.8952} C_DIS
LIN {X 58.6118,Y -87.5067,Z 103,A -60.5645,B 24.9459,C -1.6985,E1 25.0884,E2 506.2382} C_DIS
LIN {X 56.3475,Y -88.9824,Z 103,A -62.0238,B 24.9461,C -1.6961,E1 25.0849,E2 507.6984} C_DIS
LIN {X 54.1467,Y -90.3384,Z 103,A -63.4242,B 24.9462,C -1.6937,E1 25.0816,E2 509.1} C_DIS
LIN {X 51.9134,Y -91.64,Z 103,A -64.8253,B 24.9464,C -1.6913,E1 25.0782,E2 510.5025} C_DIS
LIN {X 49.6488,Y -92.8864,Z 103,A -66.226,B 24.9465,C -1.6891,E1 25.0748,E2 511.9044} C_DIS
LIN {X 47.3543,Y -94.0769,Z 103,A -67.6271,B 24.9467,C -1.687,E1 25.0713,E2 513.3068} C_DIS
LIN {X 45.0313,Y -95.2107,Z 103,A -69.0286,B 24.9468,C -1.6849,E1 25.0677,E2 514.7095} C_DIS
LIN {X 42.7886,Y -96.2387,Z 103,A -70.3552,B 24.9468,C -1.6835,E1 25.0644,E2 516.0362} C_DIS
LIN {X 40.3053,Y -97.3056,Z 103,A -71.8318,B 24.947,C -1.681,E1 25.0606,E2 517.515} C_DIS
LIN {X 37.9052,Y -98.2654,Z 103,A -73.2338,B 24.9472,C -1.6792,E1 25.0569,E2 518.9182} C_DIS
LIN {X 35.4822,Y -99.1661,Z 103,A -74.6362,B 24.9472,C -1.6775,E1 25.0532,E2 520.3216} C_DIS
LIN {X 33.1495,Y -99.9693,Z 103,A -75.9747,B 24.9474,C -1.676,E1 25.0497,E2 521.6612} C_DIS
LIN {X 30.5736,Y -100.7876,Z 103,A -77.4411,B 24.9474,C -1.6744,E1 25.0458,E2 523.1286} C_DIS
LIN {X 28.0909,Y -101.5076,Z 103,A -78.8441,B 24.9476,C -1.673,E1 25.042,E2 524.5327} C_DIS
LIN {X 25.827,Y -102.1059,Z 103,A -80.1257,B 24.9476,C -1.6714,E1 25.0385,E2 525.8161} C_DIS
LIN {X 23.0764,Y -102.7637,Z 103,A -81.6505,B 24.9477,C -1.6704,E1 25.0344,E2 527.341} C_DIS
LIN {X 20.6629,Y -103.2754,Z 103,A -82.9904,B 24.9477,C -1.6694,E1 25.0307,E2 528.6818} C_DIS
LIN {X 18.5589,Y -103.6728,Z 103,A -84.2241,B 24.948,C -1.6657,E1 25.0273,E2 529.9229} C_DIS
LIN {X 16.0353,Y -104.093,Z 103,A -85.634,B 24.9481,C -1.6639,E1 25.0234,E2 531.3355} C_DIS
LIN {X 13.0095,Y -104.5156,Z 103,A -87.2074,B 24.948,C -1.6664,E1 25.0191,E2 532.9018} C_DIS
LIN {X 10.4406,Y -104.8034,Z 103,A -88.6118,B 24.948,C -1.6656,E1 25.0152,E2 534.307} C_DIS
LIN {X 7.748,Y -105.0374,Z 103,A -90.0754,B 24.948,C -1.6652,E1 25.0111,E2 535.771} C_DIS
LIN {X 3.9944,Y -105.2464,Z 103,A -92.1229,B 24.948,C -1.6643,E1 25.0054,E2 537.8199} C_DIS
LIN {X 0.7313,Y -105.3176,Z 103,A -93.5559,B 24.9473,C -1.6774,E1 25.0015,E2 539.2216} C_DIS
Enddeposition()
LIN {X 0.7313,Y -105.3176,Z 103,A -93.5559,B 24.9473,C -1.6774,E1 25.0015,E2 539.2216} C_DIS
Startdeposition()
$VEL.CP = VEL_PRINT
LIN {X 4.3118,Y -104.2345,Z 103,A -91.5163,B 24.946,C -1.6983,E1 25.0073,E2 537.1329} C_DIS
LIN {X 6.2818,Y -104.1355,Z 103,A -89.9598,B 24.9447,C -1.7175,E1 25.0118,E2 535.5313} C_DIS
LIN {X 9.5979,Y -103.881,Z 103,A -88.2237,B 24.9449,C -1.7149,E1 25.0166,E2 533.8025} C_DIS
LIN {X 13.3836,Y -103.4614,Z 103,A -86.2269,B 24.9451,C -1.7123,E1 25.0221,E2 531.8132} C_DIS
LIN {X 16.2567,Y -103.0495,Z 103,A -84.5107,B 24.9447,C -1.7184,E1 25.0269,E2 530.0843} C_DIS
LIN {X 19.8266,Y -102.4222,Z 103,A -82.6875,B 24.945,C -1.7133,E1 25.0318,E2 528.2754} C_DIS
LIN {X 23.4099,Y -101.663,Z 103,A -80.5958,B 24.9447,C -1.7183,E1 25.0376,E2 526.1744} C_DIS
LIN {X 26.2663,Y -100.9632,Z 103,A -79.044,B 24.9447,C -1.7174,E1 25.0418,E2 524.6271} C_DIS
LIN {X 30.9406,Y -99.6296,Z 103,A -75.9557,B 24.9434,C -1.7376,E1 25.0501,E2 521.4965} C_DIS
LIN {X 34.1295,Y -98.5837,Z 103,A -74.6347,B 24.9447,C -1.7185,E1 25.0535,E2 520.2232} C_DIS
LIN {X 38.2304,Y -97.0661,Z 103,A -72.1503,B 24.9442,C -1.7252,E1 25.06,E2 517.7284} C_DIS
LIN {X 41.7257,Y -95.6157,Z 103,A -70.1971,B 24.9444,C -1.7231,E1 25.065,E2 515.7848} C_DIS
LIN {X 44.5392,Y -94.3397,Z 103,A -68.4743,B 24.9441,C -1.7268,E1 25.0694,E2 514.0575} C_DIS
LIN {X 47.4037,Y -92.9316,Z 103,A -66.8652,B 24.9443,C -1.7238,E1 25.0734,E2 512.4598} C_DIS
LIN {X 49.5847,Y -91.7866,Z 103,A -64.4653,B 24.9413,C -1.7696,E1 25.0795,E2 509.9586} C_DIS
LIN {X 53.8608,Y -89.3451,Z 103,A -62.4933,B 24.943,C -1.744,E1 25.0841,E2 508.0532} C_DIS
LIN {X 56.5388,Y -87.6744,Z 103,A -60.2559,B 24.9414,C -1.7684,E1 25.0895,E2 505.7653} C_DIS
LIN {X 59.9442,Y -85.3834,Z 103,A -58.7356,B 24.9431,C -1.7423,E1 25.0928,E2 504.312} C_DIS
LIN {X 62.0362,Y -83.8758,Z 103,A -57.2902,B 24.9428,C -1.7464,E1 25.0961,E2 502.8619} C_DIS
LIN {X 64.6386,Y -81.8855,Z 103,A -55.4094,B 24.9424,C -1.7538,E1 25.1003,E2 500.9707} C_DIS
LIN {X 68.1051,Y -79.0272,Z 103,A -52.8463,B 24.9417,C -1.7633,E1 25.1058,E2 498.3949} C_DIS
LIN {X 70.3066,Y -77.0744,Z 103,A -51.33,B 24.9417,C -1.7629,E1 25.1089,E2 496.8858} C_DIS
LIN {X 72.6754,Y -74.8453,Z 103,A -49.6427,B 24.9417,C -1.763,E1 25.1123,E2 495.2051} C_DIS
LIN {X 74.7968,Y -72.7258,Z 103,A -47.7314,B 24.9407,C -1.7782,E1 25.1161,E2 493.2662} C_DIS
LIN {X 78.5435,Y -68.6608,Z 103,A -45.1027,B 24.9414,C -1.7688,E1 25.1209,E2 490.6714} C_DIS
LIN {X 80.4668,Y -66.3974,Z 103,A -43.3137,B 24.9406,C -1.7797,E1 25.1242,E2 488.8648} C_DIS
LIN {X 82.5461,Y -63.793,Z 103,A -41.5972,B 24.9406,C -1.7797,E1 25.1271,E2 487.1561} C_DIS
LIN {X 84.5538,Y -61.1101,Z 103,A -38.9259,B 24.9379,C -1.8201,E1 25.1317,E2 484.4025} C_DIS
LIN {X 87.0699,Y -57.4649,Z 103,A -37.5595,B 24.9405,C -1.7816,E1 25.1336,E2 483.1336} C_DIS
LIN {X 88.2103,Y -55.7009,Z 103,A -35.8805,B 24.9388,C -1.8071,E1 25.1362,E2 481.4029} C_DIS
LIN {X 90.2853,Y -52.2691,Z 103,A -33.7868,B 24.9387,C -1.8089,E1 25.1392,E2 479.3159} C_DIS
LIN {X 92.026,Y -49.1409,Z 103,A -31.8243,B 24.9383,C -1.8145,E1 25.1418,E2 477.3503} C_DIS
LIN {X 93.8,Y -45.6643,Z 103,A -29.9432,B 24.9386,C -1.8098,E1 25.1441,E2 475.4904} C_DIS
LIN {X 95.2412,Y -42.5747,Z 103,A -27.8512,B 24.9376,C -1.8248,E1 25.1466,E2 473.3743} C_DIS
LIN {X 97.5279,Y -37.0366,Z 103,A -24.6628,B 24.9372,C -1.8306,E1 25.1499,E2 470.19} C_DIS
LIN {X 98.8209,Y -33.434,Z 103,A -22.6681,B 24.9371,C -1.8326,E1 25.1517,E2 468.2018} C_DIS
LIN {X 99.8165,Y -30.338,Z 103,A -20.6861,B 24.9361,C -1.8465,E1 25.1534,E2 466.1981} C_DIS
LIN {X 100.9146,Y -26.4553,Z 103,A -18.5256,B 24.9358,C -1.8512,E1 25.155,E2 464.039} C_DIS
LIN {X 101.8185,Y -22.7296,Z 103,A -16.5129,B 24.9356,C -1.854,E1 25.1562,E2 462.0315} C_DIS
LIN {X 102.617,Y -18.7947,Z 103,A -14.5755,B 24.9359,C -1.8496,E1 25.1573,E2 460.1155} C_DIS
LIN {X 103.0015,Y -16.5672,Z 103,A -12.9944,B 24.9346,C -1.8681,E1 25.158,E2 458.5003} C_DIS
LIN {X 103.502,Y -13.0706,Z 103,A -11.0683,B 24.9342,C -1.8738,E1 25.1587,E2 456.5721} C_DIS
LIN {X 103.8679,Y -9.7405,Z 103,A -9.3492,B 24.9342,C -1.8746,E1 25.1592,E2 454.8613} C_DIS
LIN {X 104.131,Y -6.3626,Z 103,A -7.2294,B 24.9329,C -1.8917,E1 25.1596,E2 452.7138} C_DIS
LIN {X 104.312,Y -1.5812,Z 103,A -5.1179,B 24.9339,C -1.8782,E1 25.1598,E2 450.6467} C_DIS
LIN {X 104.3208,Y 0.7696,Z 103,A -3.5685,B 24.9328,C -1.8933,E1 25.1598,E2 449.0708} C_DIS
LIN {X 104.2171,Y 4.7148,Z 103,A -1.3768,B 24.9322,C -1.9013,E1 25.1595,E2 446.8732} C_DIS
LIN {X 103.9697,Y 8.5886,Z 103,A 0.673,B 24.932,C -1.9047,E1 25.1591,E2 444.8277} C_DIS
LIN {X 103.6133,Y 12.1524,Z 103,A 2.5903,B 24.9317,C -1.9088,E1 25.1586,E2 442.912} C_DIS
LIN {X 103.1524,Y 15.5916,Z 103,A 4.5988,B 24.9309,C -1.9192,E1 25.1578,E2 440.8907} C_DIS
LIN {X 102.6576,Y 18.5694,Z 103,A 6.1897,B 24.9308,C -1.9216,E1 25.157,E2 439.3036} C_DIS
LIN {X 102.08,Y 21.5262,Z 103,A 7.9069,B 24.9302,C -1.9294,E1 25.156,E2 437.5779} C_DIS
LIN {X 101.3668,Y 24.6609,Z 103,A 9.6781,B 24.9298,C -1.9351,E1 25.1549,E2 435.8035} C_DIS
LIN {X 100.3523,Y 28.5099,Z 103,A 11.6803,B 24.9298,C -1.934,E1 25.1534,E2 433.8154} C_DIS
LIN {X 99.4508,Y 31.5171,Z 103,A 13.6236,B 24.9288,C -1.9485,E1 25.1518,E2 431.849} C_DIS
LIN {X 98.2055,Y 35.205,Z 103,A 15.5573,B 24.929,C -1.9462,E1 25.15,E2 429.9316} C_DIS
LIN {X 96.5106,Y 39.613,Z 103,A 18.0763,B 24.9287,C -1.9507,E1 25.1475,E2 427.4161} C_DIS
LIN {X 95.0026,Y 43.104,Z 103,A 20.1403,B 24.9283,C -1.9556,E1 25.1451,E2 425.3517} C_DIS
LIN {X 93.5295,Y 46.2129,Z 103,A 22.1242,B 24.9276,C -1.9649,E1 25.1427,E2 423.3564} C_DIS
LIN {X 91.7774,Y 49.6015,Z 103,A 24.2283,B 24.9272,C -1.9711,E1 25.1399,E2 421.2488} C_DIS
LIN {X 89.803,Y 53.0925,Z 103,A 26.3679,B 24.9269,C -1.9744,E1 25.137,E2 419.1125} C_DIS
LIN {X 88.4118,Y 55.3784,Z 103,A 27.7984,B 24.9267,C -1.9766,E1 25.1349,E2 417.684} C_DIS
LIN {X 86.3772,Y 58.5009,Z 103,A 29.7423,B 24.9267,C -1.9776,E1 25.1319,E2 415.7475} C_DIS
LIN {X 84.5498,Y 61.1157,Z 103,A 31.5147,B 24.9263,C -1.9828,E1 25.129,E2 413.9714} C_DIS
LIN {X 81.9359,Y 64.5749,Z 103,A 33.6431,B 24.9266,C -1.9782,E1 25.1255,E2 411.8641} C_DIS
LIN {X 79.8244,Y 67.1703,Z 103,A 35.7117,B 24.9256,C -1.992,E1 25.1217,E2 409.7723} C_DIS
LIN {X 78.1769,Y 69.0806,Z 103,A 37.7353,B 24.9234,C -2.0217,E1 25.1179,E2 407.6876} C_DIS
LIN {X 75.5676,Y 71.9258,Z 103,A 39.195,B 24.9251,C -1.999,E1 25.1152,E2 406.288} C_DIS
LIN {X 72.3643,Y 75.1452,Z 103,A 41.9846,B 24.9238,C -2.0165,E1 25.1096,E2 403.4687} C_DIS
LIN {X 69.9294,Y 77.4176,Z 103,A 43.6018,B 24.9241,C -2.0115,E1 25.1063,E2 401.8701} C_DIS
LIN {X 67.2876,Y 79.7245,Z 103,A 45.8903,B 24.9227,C -2.0301,E1 25.1014,E2 399.5463} C_DIS
LIN {X 64.4201,Y 82.0582,Z 103,A 47.7107,B 24.9231,C -2.0252,E1 25.0974,E2 397.7443} C_DIS
LIN {X 60.9745,Y 84.6506,Z 103,A 49.7204,B 24.9239,C -2.0147,E1 25.093,E2 395.7666} C_DIS
LIN {X 58.4464,Y 86.4142,Z 103,A 51.4626,B 24.9235,C -2.0196,E1 25.089,E2 394.0189} C_DIS
LIN {X 55.8599,Y 88.1102,Z 103,A 53.2636,B 24.923,C -2.0264,E1 25.0847,E2 392.2076} C_DIS
LIN {X 53.4799,Y 89.574,Z 103,A 54.8812,B 24.9226,C -2.032,E1 25.0808,E2 390.5817} C_DIS
LIN {X 50.2143,Y 91.445,Z 103,A 56.7249,B 24.923,C -2.0259,E1 25.0764,E2 388.7579} C_DIS
LIN {X 47.5207,Y 92.8718,Z 103,A 58.5523,B 24.9224,C -2.0343,E1 25.0718,E2 386.9158} C_DIS
LIN {X 44.9135,Y 94.1608,Z 103,A 60.2053,B 24.9221,C -2.0385,E1 25.0677,E2 385.2571} C_DIS
LIN {X 41.7441,Y 95.6076,Z 103,A 62.071,B 24.9221,C -2.0388,E1 25.0629,E2 383.3955} C_DIS
LIN {X 38.0563,Y 97.1345,Z 103,A 64.5216,B 24.9211,C -2.0514,E1 25.0565,E2 380.9205} C_DIS
LIN {X 33.7479,Y 98.715,Z 103,A 66.7549,B 24.9218,C -2.0421,E1 25.0507,E2 378.7137} C_DIS
LIN {X 30.8772,Y 99.6493,Z 103,A 68.413,B 24.9217,C -2.0434,E1 25.0463,E2 377.0555} C_DIS
LIN {X 27.0139,Y 100.7654,Z 103,A 70.7096,B 24.9213,C -2.0484,E1 25.0401,E2 374.7509} C_DIS
LIN {X 23.118,Y 101.7304,Z 103,A 72.7825,B 24.9216,C -2.0444,E1 25.0345,E2 372.6904} C_DIS
LIN {X 19.5684,Y 102.4719,Z 103,A 74.7221,B 24.9217,C -2.0433,E1 25.0292,E2 370.7559} C_DIS
LIN {X 16.6068,Y 102.9949,Z 103,A 76.4645,B 24.9214,C -2.0474,E1 25.0244,E2 369.0055} C_DIS
LIN {X 13.7138,Y 103.4186,Z 103,A 78.1119,B 24.9212,C -2.0494,E1 25.0198,E2 367.3548} C_DIS
LIN {X 9.8333,Y 103.8593,Z 103,A 80.2769,B 24.9212,C -2.0505,E1 25.0138,E2 365.1885} C_DIS
LIN {X 6.5308,Y 104.1201,Z 103,A 82.1214,B 24.9211,C -2.0515,E1 25.0086,E2 363.3425} C_DIS
LIN {X 2.9515,Y 104.282,Z 103,A 84.074,B 24.9211,C -2.0508,E1 25.0032,E2 361.3922} C_DIS
LIN {X -0.8006,Y 104.3205,Z 103,A 86.1411,B 24.9211,C -2.0506,E1 24.9974,E2 359.3255} C_DIS
LIN {X -4.2525,Y 104.237,Z 103,A 87.9697,B 24.9214,C -2.0474,E1 24.9923,E2 357.5042} C_DIS
LIN {X -7.1976,Y 104.075,Z 103,A 89.5521,B 24.9216,C -2.0453,E1 24.9879,E2 355.9262} C_DIS
LIN {X -10.8175,Y 103.7611,Z 103,A 91.5514,B 24.9216,C -2.0445,E1 24.9824,E2 353.9279} C_DIS
LIN {X -13.8648,Y 103.3991,Z 103,A 93.3343,B 24.9214,C -2.0472,E1 24.9774,E2 352.1373} C_DIS
LIN {X -17.7552,Y 102.803,Z 103,A 95.3175,B 24.9221,C -2.0389,E1 24.972,E2 350.172} C_DIS
LIN {X -21.9576,Y 101.9869,Z 103,A 97.4957,B 24.9227,C -2.0304,E1 24.9661,E2 348.0114} C_DIS
LIN {X -25.3916,Y 101.188,Z 103,A 99.7715,B 24.9219,C -2.0414,E1 24.9598,E2 345.7065} C_DIS
LIN {X -28.6531,Y 100.3117,Z 103,A 101.5281,B 24.9223,C -2.0357,E1 24.9551,E2 343.9606} C_DIS
LIN {X -31.1703,Y 99.5584,Z 103,A 102.9925,B 24.9223,C -2.0349,E1 24.9512,E2 342.4956} C_DIS
LIN {X -35.3093,Y 98.1675,Z 103,A 105.2399,B 24.923,C -2.0263,E1 24.9453,E2 340.2644} C_DIS
LIN {X -37.7665,Y 97.2483,Z 103,A 107.2472,B 24.9215,C -2.0456,E1 24.94,E2 338.2069} C_DIS
LIN {X -42.5152,Y 95.268,Z 103,A 109.8375,B 24.9225,C -2.0326,E1 24.9334,E2 335.6414} C_DIS
LIN {X -46.0749,Y 93.5979,Z 103,A 111.8697,B 24.9231,C -2.0245,E1 24.9283,E2 333.6233} C_DIS
LIN {X -50.7283,Y 91.1595,Z 103,A 114.7623,B 24.9235,C -2.0199,E1 24.9212,E2 330.7337} C_DIS
LIN {X -52.8395,Y 89.9525,Z 103,A 116.0803,B 24.9237,C -2.0168,E1 24.918,E2 329.4189} C_DIS
LIN {X -54.9518,Y 88.6782,Z 103,A 117.3173,B 24.9242,C -2.01,E1 24.9151,E2 328.1944} C_DIS
LIN {X -56.7423,Y 87.5438,Z 103,A 118.5222,B 24.9243,C -2.0092,E1 24.9123,E2 326.9874} C_DIS
LIN {X -59.3197,Y 85.8175,Z 103,A 120.2164,B 24.9246,C -2.0055,E1 24.9084,E2 325.2963} C_DIS
LIN {X -61.9099,Y 83.9683,Z 103,A 122.0732,B 24.9246,C -2.0059,E1 24.9042,E2 323.432} C_DIS
LIN {X -64.467,Y 82.0212,Z 103,A 123.9485,B 24.9246,C -2.0062,E1 24.9,E2 321.5493} C_DIS
LIN {X -66.9346,Y 80.0204,Z 103,A 125.5524,B 24.9252,C -1.9972,E1 24.8966,E2 319.9607} C_DIS
LIN {X -69.4609,Y 77.837,Z 103,A 127.5172,B 24.9252,C -1.9978,E1 24.8924,E2 317.9866} C_DIS
LIN {X -72.2633,Y 75.2425,Z 103,A 129.5658,B 24.9257,C -1.9911,E1 24.8883,E2 315.9457} C_DIS
LIN {X -74.5999,Y 72.9283,Z 103,A 131.6323,B 24.9253,C -1.9961,E1 24.8842,E2 313.8583} C_DIS
LIN {X -77.6421,Y 69.6787,Z 103,A 133.8742,B 24.9263,C -1.9827,E1 24.88,E2 311.6386} C_DIS
LIN {X -79.4879,Y 67.5653,Z 103,A 135.3725,B 24.9267,C -1.9771,E1 24.8773,E2 310.1467} C_DIS
LIN {X -81.8069,Y 64.7381,Z 103,A 137.4306,B 24.927,C -1.9737,E1 24.8737,E2 308.0873} C_DIS
LIN {X -84.412,Y 61.3039,Z 103,A 139.7137,B 24.9277,C -1.9642,E1 24.8699,E2 305.8158} C_DIS
LIN {X -86.201,Y 58.7613,Z 103,A 141.6042,B 24.9275,C -1.9661,E1 24.8669,E2 303.9115} C_DIS
LIN {X -87.8008,Y 56.3419,Z 103,A 143.1498,B 24.928,C -1.9599,E1 24.8645,E2 302.3728} C_DIS
LIN {X -89.8791,Y 52.9638,Z 103,A 145.3049,B 24.9285,C -1.9528,E1 24.8614,E2 300.2235} C_DIS
LIN {X -91.5514,Y 50.0183,Z 103,A 147.8721,B 24.927,C -1.9728,E1 24.8579,E2 297.595} C_DIS
LIN {X -93.5489,Y 46.1739,Z 103,A 149.4498,B 24.9297,C -1.9369,E1 24.856,E2 296.0944} C_DIS
LIN {X -94.682,Y 43.8038,Z 103,A 151.5743,B 24.9282,C -1.957,E1 24.8534,E2 293.9104} C_DIS
LIN {X -96.2011,Y 40.3579,Z 103,A 153.2152,B 24.9298,C -1.9354,E1 24.8517,E2 292.3122} C_DIS
LIN {X -97.487,Y 37.1445,Z 103,A 155.0382,B 24.9304,C -1.9267,E1 24.8499,E2 290.4994} C_DIS
LIN {X -98.8862,Y 33.2404,Z 103,A 157.5507,B 24.9304,C -1.928,E1 24.8475,E2 287.9696} C_DIS
LIN {X -100.9373,Y 26.3671,Z 103,A 161.7216,B 24.9306,C -1.9239,E1 24.8444,E2 283.7845} C_DIS
LIN {X -101.727,Y 23.1329,Z 103,A 162.9451,B 24.9326,C -1.8964,E1 24.8436,E2 282.6192} C_DIS
LIN {X -102.3056,Y 20.4273,Z 103,A 164.7843,B 24.9321,C -1.9029,E1 24.8426,E2 280.7537} C_DIS
LIN {X -102.9957,Y 16.6025,Z 103,A 166.7176,B 24.9331,C -1.8889,E1 24.8417,E2 278.8424} C_DIS
LIN {X -103.4166,Y 13.7295,Z 103,A 168.3132,B 24.9335,C -1.8838,E1 24.8411,E2 277.2494} C_DIS
LIN {X -103.8224,Y 10.2326,Z 103,A 170.3418,B 24.9337,C -1.8809,E1 24.8404,E2 275.2156} C_DIS
LIN {X -104.1149,Y 6.608,Z 103,A 172.2365,B 24.9344,C -1.8708,E1 24.8401,E2 273.3335} C_DIS
LIN {X -104.2554,Y 3.8175,Z 103,A 173.8196,B 24.9346,C -1.8676,E1 24.8399,E2 271.7486} C_DIS
LIN {X -104.3226,Y 0.4853,Z 103,A 175.8135,B 24.9346,C -1.8676,E1 24.8398,E2 269.7428} C_DIS
LIN {X -104.2935,Y -2.5785,Z 103,A 177.5869,B 24.9348,C -1.8653,E1 24.8398,E2 267.9641} C_DIS
LIN {X -104.141,Y -6.1829,Z 103,A 179.3761,B 24.9357,C -1.8521,E1 24.8401,E2 266.1955} C_DIS
LIN {X -103.975,Y -8.5226,Z 103,A -179.2567,B 24.9357,C -1.8508,E1 24.8404,E2 264.8232} C_DIS
LIN {X -103.6143,Y -12.1437,Z 103,A -177.2378,B 24.9362,C -1.8452,E1 24.841,E2 262.8056} C_DIS
LIN {X -102.8938,Y -17.2118,Z 103,A -174.5252,B 24.937,C -1.8328,E1 24.8422,E2 260.1065} C_DIS
LIN {X -102.3983,Y -19.9508,Z 103,A -172.7828,B 24.9368,C -1.8356,E1 24.8431,E2 258.347} C_DIS
LIN {X -101.6633,Y -23.4088,Z 103,A -171.1056,B 24.9379,C -1.8202,E1 24.8441,E2 256.6969} C_DIS
LIN {X -100.264,Y -28.8214,Z 103,A -167.9157,B 24.9383,C -1.815,E1 24.8464,E2 253.5007} C_DIS
LIN {X -99.3567,Y -31.8079,Z 103,A -165.9907,B 24.9381,C -1.8174,E1 24.848,E2 251.5589} C_DIS
LIN {X -98.2702,Y -35.0231,Z 103,A -164.0947,B 24.9384,C -1.813,E1 24.8497,E2 249.6626} C_DIS
LIN {X -97.0932,Y -38.1614,Z 103,A -162.3832,B 24.9391,C -1.8029,E1 24.8514,E2 247.9656} C_DIS
LIN {X -95.1813,Y -42.7076,Z 103,A -159.7144,B 24.9397,C -1.7937,E1 24.8543,E2 245.3041} C_DIS
LIN {X -93.9009,Y -45.4544,Z 103,A -157.9452,B 24.9397,C -1.7928,E1 24.8565,E2 243.5274} C_DIS
LIN {X -91.9101,Y -49.3569,Z 103,A -155.7358,B 24.9407,C -1.779,E1 24.8593,E2 241.339} C_DIS
LIN {X -90.3817,Y -52.1014,Z 103,A -153.883,B 24.9407,C -1.779,E1 24.8618,E2 239.4766} C_DIS
LIN {X -88.6216,Y -55.0424,Z 103,A -152.1469,B 24.9414,C -1.7687,E1 24.8643,E2 237.7561} C_DIS
LIN {X -87.0559,Y -57.4862,Z 103,A -150.2579,B 24.9409,C -1.7753,E1 24.8672,E2 235.8418} C_DIS
LIN {X -84.9175,Y -60.6004,Z 103,A -148.2385,B 24.9414,C -1.7681,E1 24.8705,E2 233.8297} C_DIS
LIN {X -82.7993,Y -63.4644,Z 103,A -146.3753,B 24.942,C -1.7598,E1 24.8736,E2 231.9771} C_DIS
LIN {X -80.748,Y -66.0558,Z 103,A -144.5374,B 24.9422,C -1.7563,E1 24.8768,E2 230.139} C_DIS
LIN {X -76.4401,Y -70.997,Z 103,A -140.9402,B 24.9427,C -1.748,E1 24.8834,E2 226.5455} C_DIS
LIN {X -74.7231,Y -72.8022,Z 103,A -139.3172,B 24.9423,C -1.7544,E1 24.8866,E2 224.9001} C_DIS
LIN {X -72.4558,Y -75.057,Z 103,A -137.6303,B 24.9427,C -1.7482,E1 24.89,E2 223.2211} C_DIS
LIN {X -70.0176,Y -77.3386,Z 103,A -135.9528,B 24.9433,C -1.7387,E1 24.8934,E2 221.5595} C_DIS
LIN {X -67.21,Y -79.79,Z 103,A -133.7178,B 24.9431,C -1.7417,E1 24.8981,E2 219.3085} C_DIS
LIN {X -64.6979,Y -81.8387,Z 103,A -131.9814,B 24.9435,C -1.7368,E1 24.9019,E2 217.5773} C_DIS
LIN {X -62.2925,Y -83.6853,Z 103,A -130.1953,B 24.9434,C -1.7384,E1 24.9059,E2 215.781} C_DIS
LIN {X -59.1899,Y -85.9077,Z 103,A -128.2134,B 24.9439,C -1.7306,E1 24.9104,E2 213.8109} C_DIS
LIN {X -56.8851,Y -87.4521,Z 103,A -126.7253,B 24.9441,C -1.7268,E1 24.9139,E2 212.3269} C_DIS
LIN {X -54.0033,Y -89.2585,Z 103,A -124.968,B 24.9446,C -1.7199,E1 24.918,E2 210.5806} C_DIS
LIN {X -51.5073,Y -90.7231,Z 103,A -123.1216,B 24.9441,C -1.7273,E1 24.9226,E2 208.7109} C_DIS
LIN {X -48.237,Y -92.5028,Z 103,A -121.0963,B 24.9443,C -1.7239,E1 24.9275,E2 206.6882} C_DIS
LIN {X -45.0621,Y -94.0894,Z 103,A -119.2441,B 24.9447,C -1.7179,E1 24.9322,E2 204.8455} C_DIS
LIN {X -42.5665,Y -95.2449,Z 103,A -117.5901,B 24.9445,C -1.7216,E1 24.9364,E2 203.1785} C_DIS
LIN {X -38.0867,Y -97.1226,Z 103,A -115.0328,B 24.9449,C -1.7147,E1 24.943,E2 200.632} C_DIS
LIN {X -34.8801,Y -98.3204,Z 103,A -113.0314,B 24.9447,C -1.7177,E1 24.9483,E2 198.6193} C_DIS
LIN {X -31.3855,Y -99.4915,Z 103,A -111.0321,B 24.9449,C -1.7152,E1 24.9536,E2 196.6224} C_DIS
LIN {X -27.8228,Y -100.5469,Z 103,A -109.1596,B 24.9454,C -1.7073,E1 24.9586,E2 194.7657} C_DIS
LIN {X -24.7692,Y -101.3404,Z 103,A -107.277,B 24.9451,C -1.7121,E1 24.9637,E2 192.8689} C_DIS
LIN {X -20.9151,Y -102.2054,Z 103,A -105.1849,B 24.9453,C -1.7081,E1 24.9694,E2 190.7837} C_DIS
LIN {X -17.7328,Y -102.8067,Z 103,A -103.5243,B 24.9457,C -1.7029,E1 24.9739,E2 189.1339} C_DIS
LIN {X -13.7645,Y -103.4121,Z 103,A -101.2757,B 24.9456,C -1.7041,E1 24.9801,E2 186.8805} C_DIS
LIN {X -10.5178,Y -103.7925,Z 103,A -99.3482,B 24.9453,C -1.7091,E1 24.9855,E2 184.94} C_DIS
LIN {X -6.9292,Y -104.0932,Z 103,A -97.423,B 24.9453,C -1.707,E1 24.9909,E2 183.019} C_DIS
LIN {X -3.2646,Y -104.2724,Z 103,A -95.3339,B 24.9452,C -1.7101,E1 24.9967,E2 180.9221} C_DIS
LIN {X 0.0858,Y -104.3249,Z 103,A -92.882,B 24.9436,C -1.7349,E1 25.0038,E2 178.4115} C_DIS
LIN {X 0.0858,Y -104.3249,Z 103,A -92.882,B 24.9436,C -1.7349,E1 25.0038,E2 178.4115} C_DIS
Enddeposition()
LIN {X 0.6967,Y -103.3193,Z 103,A -93.3201,B 24.9445,C -1.7215,E1 25.0024,E2 178.8813} C_DIS
Startdeposition()
$VEL.CP = VEL_PRINT
LIN {X -1.9029,Y -103.3086,Z 103,A -95.505,B 24.9463,C -1.6922,E1 24.9961,E2 181.1357} C_DIS
LIN {X -5.4702,Y -103.1815,Z 103,A -97.5226,B 24.9464,C -1.6905,E1 24.9905,E2 183.1577} C_DIS
LIN {X -9.1304,Y -102.9226,Z 103,A -99.5054,B 24.9464,C -1.6926,E1 24.985,E2 185.1364} C_DIS
LIN {X -12.0262,Y -102.6239,Z 103,A -101.1669,B 24.9464,C -1.691,E1 24.9804,E2 186.8028} C_DIS
LIN {X -15.693,Y -102.1275,Z 103,A -103.1925,B 24.9464,C -1.6924,E1 24.9748,E2 188.8265} C_DIS
LIN {X -19.9881,Y -101.3754,Z 103,A -105.7156,B 24.9465,C -1.6893,E1 24.9678,E2 191.3598} C_DIS
LIN {X -23.2842,Y -100.6684,Z 103,A -107.4218,B 24.9461,C -1.6964,E1 24.9632,E2 193.0512} C_DIS
LIN {X -26.1634,Y -99.9598,Z 103,A -108.9674,B 24.9458,C -1.701,E1 24.959,E2 194.5881} C_DIS
LIN {X -28.6715,Y -99.2699,Z 103,A -111.1519,B 24.9475,C -1.6742,E1 24.953,E2 196.8399} C_DIS
LIN {X -32.4158,Y -98.1117,Z 103,A -112.8464,B 24.9462,C -1.6937,E1 24.9486,E2 198.4911} C_DIS
LIN {X -39.308,Y -95.5579,Z 103,A -116.9425,B 24.946,C -1.6967,E1 24.9379,E2 202.5885} C_DIS
LIN {X -42.5066,Y -94.1779,Z 103,A -118.5336,B 24.9451,C -1.7115,E1 24.9339,E2 204.1483} C_DIS
LIN {X -46.0344,Y -92.5048,Z 103,A -120.9046,B 24.9454,C -1.7064,E1 24.9279,E2 206.5375} C_DIS
LIN {X -48.9566,Y -90.9926,Z 103,A -122.8177,B 24.9454,C -1.7055,E1 24.9232,E2 208.458} C_DIS
LIN {X -51.5517,Y -89.5473,Z 103,A -124.7545,B 24.946,C -1.6972,E1 24.9184,E2 210.4202} C_DIS
LIN {X -55.7267,Y -87.0105,Z 103,A -127.1199,B 24.945,C -1.7139,E1 24.9129,E2 212.7535} C_DIS
LIN {X -59.6025,Y -84.4043,Z 103,A -129.6705,B 24.9446,C -1.7195,E1 24.907,E2 215.2992} C_DIS
LIN {X -62.4255,Y -82.338,Z 103,A -131.6194,B 24.9444,C -1.7226,E1 24.9026,E2 217.2478} C_DIS
LIN {X -64.4284,Y -80.7805,Z 103,A -133.3027,B 24.9449,C -1.7151,E1 24.8989,E2 218.9552} C_DIS
LIN {X -67.4762,Y -78.2524,Z 103,A -135.3634,B 24.9443,C -1.7242,E1 24.8945,E2 221.0022} C_DIS
LIN {X -70.2236,Y -75.797,Z 103,A -137.4451,B 24.9441,C -1.7269,E1 24.8902,E2 223.0859} C_DIS
LIN {X -72.5995,Y -73.5228,Z 103,A -139.2341,B 24.9438,C -1.732,E1 24.8867,E2 224.8702} C_DIS
LIN {X -75.2333,Y -70.8254,Z 103,A -141.1439,B 24.9431,C -1.743,E1 24.883,E2 226.762} C_DIS
LIN {X -77.4752,Y -68.3679,Z 103,A -143.5242,B 24.944,C -1.728,E1 24.8785,E2 229.1886} C_DIS
LIN {X -80.2535,Y -65.082,Z 103,A -145.4709,B 24.9427,C -1.7492,E1 24.8751,E2 231.0937} C_DIS
LIN {X -81.7065,Y -63.2486,Z 103,A -147.3017,B 24.9437,C -1.7334,E1 24.8719,E2 232.9709} C_DIS
LIN {X -83.7843,Y -60.4715,Z 103,A -148.8431,B 24.9425,C -1.7517,E1 24.8694,E2 234.4763} C_DIS
LIN {X -85.7577,Y -57.6371,Z 103,A -150.778,B 24.9422,C -1.7558,E1 24.8664,E2 236.4109} C_DIS
LIN {X -88.4577,Y -53.4005,Z 103,A -153.6233,B 24.9419,C -1.761,E1 24.8621,E2 239.2583} C_DIS
LIN {X -90.2013,Y -50.3986,Z 103,A -155.4125,B 24.9412,C -1.771,E1 24.8597,E2 241.033} C_DIS
LIN {X -92.7679,Y -45.5037,Z 103,A -158.4155,B 24.9405,C -1.7816,E1 24.8559,E2 244.0268} C_DIS
LIN {X -95.4988,Y -39.4532,Z 103,A -162.4126,B 24.9405,C -1.781,E1 24.8513,E2 248.0473} C_DIS
LIN {X -97.0258,Y -35.5287,Z 103,A -164.5181,B 24.9395,C -1.796,E1 24.8493,E2 250.129} C_DIS
LIN {X -98.0732,Y -32.5299,Z 103,A -166.467,B 24.9396,C -1.7946,E1 24.8475,E2 252.0923} C_DIS
LIN {X -99.1783,Y -28.9849,Z 103,A -168.3078,B 24.9387,C -1.8085,E1 24.846,E2 253.9106} C_DIS
LIN {X -100.0272,Y -25.9013,Z 103,A -171.0893,B 24.9407,C -1.7791,E1 24.844,E2 256.7784} C_DIS
LIN {X -101.1694,Y -21.002,Z 103,A -173.0581,B 24.9382,C -1.816,E1 24.8429,E2 258.6708} C_DIS
LIN {X -101.6695,Y -18.429,Z 103,A -175.3057,B 24.9397,C -1.7932,E1 24.8418,E2 260.986} C_DIS
LIN {X -102.4208,Y -13.653,Z 103,A -176.9675,B 24.9368,C -1.8368,E1 24.8411,E2 262.5538} C_DIS
LIN {X -102.8995,Y -9.38,Z 103,A -179.6272,B 24.9368,C -1.8348,E1 24.8403,E2 265.2342} C_DIS
LIN {X -103.1485,Y -6.067,Z 103,A 178.5843,B 24.9364,C -1.8426,E1 24.84,E2 267.015} C_DIS
LIN {X -103.3144,Y -1.5883,Z 103,A 175.7935,B 24.9365,C -1.84,E1 24.8398,E2 269.8287} C_DIS
LIN {X -103.2837,Y 2.9678,Z 103,A 173.454,B 24.9355,C -1.8546,E1 24.8398,E2 272.1475} C_DIS
LIN {X -103.1823,Y 5.4556,Z 103,A 171.7216,B 24.9361,C -1.8469,E1 24.8402,E2 273.9086} C_DIS
LIN {X -102.9642,Y 8.651,Z 103,A 170.4109,B 24.9345,C -1.8687,E1 24.8404,E2 275.1753} C_DIS
LIN {X -102.4867,Y 13.1444,Z 103,A 167.7643,B 24.9343,C -1.8719,E1 24.8413,E2 277.83} C_DIS
LIN {X -101.9317,Y 16.9182,Z 103,A 165.743,B 24.9336,C -1.882,E1 24.8421,E2 279.8393} C_DIS
LIN {X -101.3238,Y 20.2502,Z 103,A 163.7548,B 24.9335,C -1.8841,E1 24.8432,E2 281.8341} C_DIS
LIN {X -100.7565,Y 22.9028,Z 103,A 162.0535,B 24.9335,C -1.8822,E1 24.8442,E2 283.5502} C_DIS
LIN {X -99.7489,Y 26.9525,Z 103,A 160.1596,B 24.932,C -1.904,E1 24.8455,E2 285.4029} C_DIS
LIN {X -98.6914,Y 30.5988,Z 103,A 156.9739,B 24.9342,C -1.8735,E1 24.8482,E2 288.6798} C_DIS
LIN {X -97.1223,Y 35.2642,Z 103,A 155.0696,B 24.9316,C -1.9103,E1 24.8499,E2 290.5071} C_DIS
LIN {X -95.918,Y 38.4234,Z 103,A 153.3048,B 24.9309,C -1.9198,E1 24.8516,E2 292.259} C_DIS
LIN {X -94.3576,Y 42.1078,Z 103,A 150.888,B 24.9309,C -1.9198,E1 24.8543,E2 294.6895} C_DIS
LIN {X -92.5852,Y 45.8723,Z 103,A 148.0672,B 24.9317,C -1.9089,E1 24.8578,E2 297.5514} C_DIS
LIN {X -90.8326,Y 49.2516,Z 103,A 146.2124,B 24.9306,C -1.9239,E1 24.8602,E2 299.3801} C_DIS
LIN {X -88.4439,Y 53.4233,Z 103,A 143.8654,B 24.9292,C -1.9427,E1 24.8635,E2 301.6946} C_DIS
LIN {X -86.9511,Y 55.8193,Z 103,A 141.7988,B 24.9302,C -1.9297,E1 24.8667,E2 303.8027} C_DIS
LIN {X -85.0642,Y 58.656,Z 103,A 140.5593,B 24.9282,C -1.9575,E1 24.8685,E2 304.9819} C_DIS
LIN {X -82.0589,Y 62.7913,Z 103,A 137.4387,B 24.9283,C -1.9552,E1 24.8737,E2 308.1232} C_DIS
LIN {X -79.0205,Y 66.5761,Z 103,A 134.6464,B 24.9281,C -1.9587,E1 24.8787,E2 310.9201} C_DIS
LIN {X -76.4696,Y 69.4905,Z 103,A 132.2138,B 24.9284,C -1.9542,E1 24.8833,E2 313.3743} C_DIS
LIN {X -73.8998,Y 72.2178,Z 103,A 130.1263,B 24.9281,C -1.9589,E1 24.8873,E2 315.4596} C_DIS
LIN {X -70.5448,Y 75.4972,Z 103,A 127.895,B 24.9266,C -1.9781,E1 24.8917,E2 317.6543} C_DIS
LIN {X -68.368,Y 77.4751,Z 103,A 125.9878,B 24.9271,C -1.9721,E1 24.8958,E2 319.5835} C_DIS
LIN {X -65.3319,Y 80.0509,Z 103,A 123.3637,B 24.9278,C -1.9623,E1 24.9015,E2 322.2408} C_DIS
LIN {X -61.9166,Y 82.7203,Z 103,A 121.5604,B 24.9259,C -1.9885,E1 24.9054,E2 323.9881} C_DIS
LIN {X -56.8403,Y 86.2871,Z 103,A 118.2237,B 24.9251,C -1.9991,E1 24.913,E2 327.311} C_DIS
LIN {X -54.1107,Y 88.0259,Z 103,A 116.4891,B 24.9247,C -2.0046,E1 24.9171,E2 329.038} C_DIS
LIN {X -51.5163,Y 89.5676,Z 103,A 114.0838,B 24.9264,C -1.9814,E1 24.9231,E2 331.5055} C_DIS
LIN {X -47.9449,Y 91.5291,Z 103,A 112.3375,B 24.9247,C -2.0036,E1 24.9273,E2 333.204} C_DIS
LIN {X -44.5052,Y 93.2504,Z 103,A 110.4799,B 24.9237,C -2.0169,E1 24.9319,E2 335.0348} C_DIS
LIN {X -40.7986,Y 94.9315,Z 103,A 107.7014,B 24.9249,C -2.0014,E1 24.9391,E2 337.8568} C_DIS
LIN {X -36.8464,Y 96.5334,Z 103,A 105.6378,B 24.9238,C -2.0155,E1 24.9444,E2 339.8913} C_DIS
LIN {X -30.0514,Y 98.8612,Z 103,A 101.636,B 24.9235,C -2.0196,E1 24.955,E2 343.8909} C_DIS
LIN {X -26.6247,Y 99.8375,Z 103,A 99.6554,B 24.9234,C -2.0215,E1 24.9603,E2 345.87} C_DIS
LIN {X -23.2766,Y 100.6702,Z 103,A 97.8193,B 24.923,C -2.0261,E1 24.9652,E2 347.6976} C_DIS
LIN {X -18.3312,Y 101.687,Z 103,A 95.0049,B 24.9229,C -2.0279,E1 24.9729,E2 350.5111} C_DIS
LIN {X -15.1288,Y 102.2143,Z 103,A 93.0808,B 24.9231,C -2.0245,E1 24.9783,E2 352.4449} C_DIS
LIN {X -11.6937,Y 102.6628,Z 103,A 91.1362,B 24.9231,C -2.0248,E1 24.9837,E2 354.3902} C_DIS
LIN {X -7.9802,Y 103.0178,Z 103,A 89.1794,B 24.9227,C -2.0299,E1 24.9891,E2 356.3357} C_DIS
LIN {X -4.5107,Y 103.2276,Z 103,A 87.2347,B 24.9227,C -2.0299,E1 24.9945,E2 358.2808} C_DIS
LIN {X -0.9156,Y 103.3224,Z 103,A 85.2154,B 24.9227,C -2.0295,E1 25.0001,E2 360.3013} C_DIS
LIN {X 2.6756,Y 103.2926,Z 103,A 83.1878,B 24.9228,C -2.0284,E1 25.0058,E2 362.3312} C_DIS
LIN {X 6.3588,Y 103.1321,Z 103,A 81.097,B 24.923,C -2.0267,E1 25.0117,E2 364.4253} C_DIS
LIN {X 10.061,Y 102.8367,Z 103,A 79.2482,B 24.9224,C -2.0345,E1 25.0167,E2 366.2546} C_DIS
LIN {X 12.8433,Y 102.5257,Z 103,A 77.5579,B 24.9228,C -2.029,E1 25.0215,E2 367.9567} C_DIS
LIN {X 17.3005,Y 101.8678,Z 103,A 74.9895,B 24.9231,C -2.0256,E1 25.0286,E2 370.5307} C_DIS
LIN {X 21.0335,Y 101.163,Z 103,A 72.8904,B 24.9231,C -2.0249,E1 25.0343,E2 372.6288} C_DIS
LIN {X 23.8837,Y 100.5298,Z 103,A 71.2399,B 24.9233,C -2.0228,E1 25.0388,E2 374.2821} C_DIS
LIN {X 29.4827,Y 99.0306,Z 103,A 68.204,B 24.9229,C -2.0276,E1 25.0469,E2 377.3017} C_DIS
LIN {X 34.6467,Y 97.3453,Z 103,A 64.9371,B 24.9239,C -2.0152,E1 25.0556,E2 380.5917} C_DIS
LIN {X 38.6633,Y 95.8203,Z 103,A 62.899,B 24.923,C -2.0262,E1 25.0609,E2 382.5992} C_DIS
LIN {X 42.6653,Y 94.1064,Z 103,A 60.4046,B 24.9235,C -2.0204,E1 25.0673,E2 385.1013} C_DIS
LIN {X 45.4297,Y 92.8046,Z 103,A 58.5876,B 24.924,C -2.0135,E1 25.0719,E2 386.9299} C_DIS
LIN {X 48.3699,Y 91.3055,Z 103,A 56.9414,B 24.9236,C -2.0183,E1 25.0759,E2 388.56} C_DIS
LIN {X 51.8577,Y 89.3715,Z 103,A 54.5692,B 24.9243,C -2.0089,E1 25.0817,E2 390.9476} C_DIS
LIN {X 56.2547,Y 86.6716,Z 103,A 51.8264,B 24.9243,C -2.0091,E1 25.0882,E2 393.681} C_DIS
LIN {X 58.9014,Y 84.8935,Z 103,A 50.0502,B 24.9246,C -2.0059,E1 25.0923,E2 395.4588} C_DIS
LIN {X 61.6534,Y 82.9181,Z 103,A 47.9807,B 24.9254,C -1.995,E1 25.097,E2 397.5467} C_DIS
LIN {X 64.5383,Y 80.6934,Z 103,A 45.8821,B 24.9259,C -1.9882,E1 25.1016,E2 399.6537} C_DIS
LIN {X 67.9658,Y 77.8264,Z 103,A 43.6498,B 24.9255,C -1.9932,E1 25.1063,E2 401.8654} C_DIS
LIN {X 71.8848,Y 74.2221,Z 103,A 40.8441,B 24.9255,C -1.993,E1 25.112,E2 404.6601} C_DIS
LIN {X 73.3924,Y 72.7315,Z 103,A 38.582,B 24.9289,C -1.9471,E1 25.1166,E2 407.021} C_DIS
LIN {X 77.225,Y 68.6492,Z 103,A 36.4687,B 24.9265,C -1.9797,E1 25.1204,E2 409.048} C_DIS
LIN {X 78.9827,Y 66.6204,Z 103,A 35.0625,B 24.9265,C -1.9795,E1 25.123,E2 410.4482} C_DIS
LIN {X 81.0356,Y 64.1056,Z 103,A 32.769,B 24.9283,C -1.9553,E1 25.127,E2 412.7881} C_DIS
LIN {X 83.1366,Y 61.3575,Z 103,A 31.2826,B 24.9274,C -1.968,E1 25.1295,E2 414.2373} C_DIS
LIN {X 85.1126,Y 58.5863,Z 103,A 29.4313,B 24.9276,C -1.9647,E1 25.1324,E2 416.0874} C_DIS
LIN {X 87.003,Y 55.7385,Z 103,A 27.5327,B 24.928,C -1.9597,E1 25.1353,E2 417.9884} C_DIS
LIN {X 89.9435,Y 50.8602,Z 103,A 24.4118,B 24.9285,C -1.9527,E1 25.1398,E2 421.1097} C_DIS
LIN {X 91.6199,Y 47.7729,Z 103,A 22.3845,B 24.9291,C -1.9441,E1 25.1424,E2 423.1466} C_DIS
LIN {X 93.1001,Y 44.8182,Z 103,A 20.7473,B 24.9289,C -1.947,E1 25.1444,E2 424.7681} C_DIS
LIN {X 94.6154,Y 41.5244,Z 103,A 18.6734,B 24.9295,C -1.9387,E1 25.1468,E2 426.8506} C_DIS
LIN {X 95.7156,Y 38.9206,Z 103,A 15.9043,B 24.9334,C -1.8852,E1 25.1499,E2 429.7306} C_DIS
LIN {X 97.9239,Y 32.9726,Z 103,A 13.5992,B 24.9306,C -1.9241,E1 25.1519,E2 431.9309} C_DIS
LIN {X 98.9845,Y 29.6383,Z 103,A 10.9132,B 24.9332,C -1.8876,E1 25.1541,E2 434.6875} C_DIS
LIN {X 100.2327,Y 25.1015,Z 103,A 8.8276,B 24.9323,C -1.901,E1 25.1555,E2 436.7295} C_DIS
LIN {X 101.1471,Y 21.1108,Z 103,A 6.735,B 24.9323,C -1.9013,E1 25.1567,E2 438.8093} C_DIS
LIN {X 101.6714,Y 18.4184,Z 103,A 5.0177,B 24.9331,C -1.8884,E1 25.1576,E2 440.5469} C_DIS
LIN {X 102.3977,Y 13.8316,Z 103,A 2.6997,B 24.933,C -1.8909,E1 25.1585,E2 442.8455} C_DIS
LIN {X 102.8144,Y 10.2814,Z 103,A 0.7773,B 24.9332,C -1.8871,E1 25.1591,E2 444.7655} C_DIS
LIN {X 103.1063,Y 6.7403,Z 103,A -1.2813,B 24.9339,C -1.8771,E1 25.1595,E2 446.8355} C_DIS
LIN {X 103.2814,Y 3.0429,Z 103,A -3.23,B 24.9341,C -1.8748,E1 25.1597,E2 448.778} C_DIS
LIN {X 103.3237,Y -0.7299,Z 103,A -5.3072,B 24.9345,C -1.8687,E1 25.1597,E2 450.8572} C_DIS
LIN {X 103.2379,Y -4.2727,Z 103,A -7.2535,B 24.9349,C -1.8631,E1 25.1596,E2 452.8052} C_DIS
LIN {X 103.0301,Y -7.8261,Z 103,A -9.2173,B 24.9354,C -1.8571,E1 25.1592,E2 454.7713} C_DIS
LIN {X 102.7329,Y -11.0605,Z 103,A -11.0404,B 24.9358,C -1.8504,E1 25.1587,E2 456.5996} C_DIS
LIN {X 102.2888,Y -14.6043,Z 103,A -12.932,B 24.936,C -1.8477,E1 25.158,E2 458.4864} C_DIS
LIN {X 101.7255,Y -18.1174,Z 103,A -15.5453,B 24.9383,C -1.8148,E1 25.1567,E2 461.1619} C_DIS
LIN {X 100.9172,Y -22.182,Z 103,A -17.2744,B 24.9372,C -1.831,E1 25.1558,E2 462.8428} C_DIS
LIN {X 99.9845,Y -26.0675,Z 103,A -19.4997,B 24.9377,C -1.8235,E1 25.1542,E2 465.0728} C_DIS
LIN {X 99.0548,Y -29.4012,Z 103,A -21.2748,B 24.9377,C -1.8235,E1 25.1529,E2 466.838} C_DIS
Enddeposition()
END
